// TwinCAT 3 PLC project JOGAN
// ProgramVersion: 3.1.4020.4
// libraries:
//   Tc2_Standard, * (Beckhoff Automation GmbH)
//   Tc2_System, * (Beckhoff Automation GmbH)
//   Tc3_Module, * (Beckhoff Automation GmbH)
// project tree:
//   DUTs/ T_CURRENT_TRANSACTION.TcDUT, T_JIG_SOCKET.TcDUT
//   GVLs/ FLAG_VAR.TcGVL, INDEXING_1_VAR.TcGVL, INDEXING_2_VAR.TcGVL, INPUT_G6_VAR.TcGVL, INPUT_VAR.TcGVL, LOADER_RS4_VAR.TcGVL, LOADER_VAR.TcGVL, POWER_CONTROL.TcGVL (not stored), SORTER_RS4_VAR.TcGVL, SORTER_VAR.TcGVL, TESTER_C8_VAR.TcGVL
//   / PlcTask.TcTTO
//   POUs/ EXECUTE_FUNCTION.TcPOU, INPUT_PROG.TcPOU, MAIN.TcPOU, STQWE.TcPOU (not stored)
//   POUs/FUKUDA/ FUKUDA_MOVE.TcPOU, FUKUDA_MOVE_1.TcPOU, LOAD_FUKUDA.TcPOU, LOAD_FUKUDA_1.TcPOU (not stored), RETURN_FUKUDA.TcPOU, RETURN_FUKUDA_1.TcPOU
//   POUs/LASER/ LASER_MOVE.TcPOU, LOAD_LASER.TcPOU, LOAD_NG.TcPOU, POU.TcPOU, RETURN_LASER.TcPOU, RETURN_NG.TcPOU
//   POUs/LOADER/ INDEXING.TcPOU, INDEX_1.TcPOU (not stored), INDEXING_2.TcPOU, STRAIGHTENING_PROG_1.TcPOU, STR.TcPOU
//   POUs/ROBOT/ INPUT_G6.TcPOU, INPUT_G61.TcPOU, LOADER_RS4.TcPOU, SORTER_RS4.TcPOU
// real-time tasks:
//   TASK PlcTask: cycle T#10ms, priority 20, ADS port 350
// I/O:
//   DEVICE Device 5 (EtherCAT), AmsNetId 172.18.128.227.6.1
//     Term 1 (EK1100) [EK1100 EtherCAT Coupler (2A E-Bus)]
//       Term 2 (EL1808) [EL1808 8Ch. Dig. Input 24V, 3ms]
//       Term 3 (EL1808) [EL1808 8Ch. Dig. Input 24V, 3ms]
//       Term 4 (EL1808) [EL1808 8Ch. Dig. Input 24V, 3ms]
//       Term 5 (EL1808) [EL1808 8Ch. Dig. Input 24V, 3ms]
//       Term 6 (EL2808) [EL2808 8Ch. Dig. Output 24V, 0.5A]
//       Term 7 (EL2808) [EL2808 8Ch. Dig. Output 24V, 0.5A]
//       Term 8 (EL2808) [EL2808 8Ch. Dig. Output 24V, 0.5A]
//       Term 9 (EL2808) [EL2808 8Ch. Dig. Output 24V, 0.5A]
//       Term 10 (EL2808) [EL2808 8Ch. Dig. Output 24V, 0.5A]
//       Term 11 (EL3058) [EL3058 8Ch. Ana. Input 4-20mA]
//       Term 12 (EL1904) [EL1904, 4 Ch. Safety Input 24V, TwinSAFE]
//         modules: Module 1 (FSOES)
//       Term 13 (EL1904) [EL1904, 4 Ch. Safety Input 24V, TwinSAFE]
//         modules: Module 1 (FSOES)
//       Term 14 (EL6731) [EL6731 PROFIBUS DP Master]
//       Term 15 (EK1110) [EK1110 EtherCAT extension]
//     Term 16 (EK1100) [EK1100 EtherCAT Coupler (2A E-Bus)]
//       Term 17 (EL1808) [EL1808 8Ch. Dig. Input 24V, 3ms]
//       Term 18 (EL1808) [EL1808 8Ch. Dig. Input 24V, 3ms]
//       Term 19 (EL1808) [EL1808 8Ch. Dig. Input 24V, 3ms]
//       Term 20 (EL1808) [EL1808 8Ch. Dig. Input 24V, 3ms]
//       Term 21 (EL1808) [EL1808 8Ch. Dig. Input 24V, 3ms]
//       Term 22 (EL1808) [EL1808 8K. Dig. Eingang 24V, 3ms]
//       Term 23 (EL2808) [EL2808 8Ch. Dig. Output 24V, 0.5A]
//       Term 24 (EL2808) [EL2808 8Ch. Dig. Output 24V, 0.5A]
//       Term 25 (EL2808) [EL2808 8Ch. Dig. Output 24V, 0.5A]
//       Term 26 (EL2808) [EL2808 8Ch. Dig. Output 24V, 0.5A]
//       Term 27 (EL2808) [EL2808 8Ch. Dig. Output 24V, 0.5A]
//       Term 28 (EL2808) [EL2808 8Ch. Dig. Output 24V, 0.5A]
//       Term 29 (EL2808) [EL2808 8Ch. Dig. Output 24V, 0.5A]
//       Term 30 (EL2808) [EL2808 8Ch. Dig. Output 24V, 0.5A]
//       Term 31 (EL6731) [EL6731 PROFIBUS DP Master]
//       Term 32 (EK1110) [EK1110 EtherCAT extension]
//     Box 33 (EP2809-0021)RS4-2 [EP2809-0021 16 Ch. Dig. Output 24V, 0,5A, M8]
//     Box 34 (EP1809-0021) [EP1809-0021 16 Ch. Dig. Input 24V, 3ms, M8]
//     Box 35 (EP2809-0021)RS4-1 [EP2809-0021 16 Ch. Dig. Output 24V, 0,5A, M8]
//     Box 36 (EP2809-0021)RS4-1 [EP1809-0021 16 Ch. Dig. Input 24V, 3ms, M8]
//     Box 37 (EP1809-0021) [EP1809-0021 16 Ch. Dig. Input 24V, 3ms, M8]
//     Box 38 (EP2809-0021) G6 [EP2809-0021 16 Ch. Dig. Output 24V, 0,5A, M8]
//     Box 39 (EPSON RC700 EtherCAT Slave)G6 [EPSON RC700 EtherCAT Slave]
//     Box 40 (EPSON RC700 EtherCAT Slave)RS4-1 [EPSON RC700 EtherCAT Slave]
//     Box 40 (EPSON RC700 EtherCAT Slave)C8 [EPSON RC700 EtherCAT Slave] (disabled)
//     Box 88 (EP2339-0021) [EP2339-0021 16 Ch. Dig. Input/Output 24V, 0,5A, M8] (disabled)
//     Box 42 (EPSON RC700 EtherCAT Slave)RS4-2 [EPSON RC700 EtherCAT Slave]
//   DEVICE Device 1 (EL6731), AmsNetId 172.18.128.227.2.1
//     Box 43 (LEC-GPR1) // Vendor: SMC Corporation Revision: V1.0
//     Box 44 (AX9000T) INDEXING 1 // Vendor: CKD Corporation Revision: Version 1.000
//      // Vendor: CKD Corporation Revision: Version 1.000
//   DEVICE Device 2 (EL6731), AmsNetId 172.18.128.227.3.1
//     Box 46 (LEC-GPR1) // Vendor: SMC Corporation Revision: V1.0
// variable links:
//   JOGAN/JOGAN Instance <-> Device 1 (EL6731)/
//     PlcTask Inputs/INDEXING_2_VAR.DataByteInput2 <-> Module 1 (8 Bytes Out,8 Bytes In)/Inputs/8 Bytes Out,8 Bytes In_0_0
//     PlcTask Outputs/INDEXING_2_VAR.DataByteOutput2 <-> Module 1 (8 Bytes Out,8 Bytes In)/Outputs/8 Bytes Out,8 Bytes In_1_0
//   JOGAN/JOGAN Instance <-> Device 1 (EL6731)/Box 43 (LEC-GPR1)
//     PlcTask Inputs/INPUT_VAR.DataWordInput1 <-> Module 1 (Input 16 words)/Inputs/Input 16 words_0_0
//     PlcTask Inputs/INPUT_VAR.DataWordInput2 <-> Module 2 (Input 16 words)/Inputs/Input 16 words_0_0
//     PlcTask Inputs/INPUT_VAR.DataWordInput3 <-> Module 3 (Input 16 words)/Inputs/Input 16 words_0_0
//     PlcTask Outputs/INPUT_VAR.DataWordOutput1 <-> Module 5 (Output 16 words)/Outputs/Output 16 words_1_0
//     PlcTask Outputs/INPUT_VAR.DataWordOutput2 <-> Module 6 (Output 16 words)/Outputs/Output 16 words_1_0
//     PlcTask Outputs/INPUT_VAR.DataWordOutput3 <-> Module 7 (Output 16 words)/Outputs/Output 16 words_1_0
//     PlcTask Outputs/INPUT_VAR.DataWordOutput4 <-> Module 8 (Output 9 words)/Outputs/Output 9 words_1_0
//   JOGAN/JOGAN Instance <-> Device 1 (EL6731)/Box 44 (AX9000T) INDEXING 1
//     PlcTask Inputs/INDEXING_1_VAR.DataByteInput <-> Module 2 (8 Bytes Out,8 Bytes In)/Inputs/8 Bytes Out,8 Bytes In_0_0
//     PlcTask Outputs/INDEXING_1_VAR.DataByteOutput <-> Module 2 (8 Bytes Out,8 Bytes In)/Outputs/8 Bytes Out,8 Bytes In_1_0
//   JOGAN/JOGAN Instance <-> Device 2 (EL6731)/Box 46 (LEC-GPR1)
//     PlcTask Inputs/SORTER_VAR.DataWordInput1 <-> Module 1 (Input 16 words)/Inputs/Input 16 words_0_0
//     PlcTask Inputs/SORTER_VAR.DataWordInput2 <-> Module 2 (Input 16 words)/Inputs/Input 16 words_0_0
//     PlcTask Inputs/SORTER_VAR.DataWordInput3 <-> Module 3 (Input 16 words)/Inputs/Input 16 words_0_0
//     PlcTask Inputs/SORTER_VAR.DataWordInput4 <-> Module 4 (Input 9 words)/Inputs/Input 9 words_0_0
//     PlcTask Outputs/SORTER_VAR.DataWordOutput1 <-> Module 5 (Output 16 words)/Outputs/Output 16 words_1_0
//     PlcTask Outputs/SORTER_VAR.DataWordOutput2 <-> Module 6 (Output 16 words)/Outputs/Output 16 words_1_0
//     PlcTask Outputs/SORTER_VAR.DataWordOutput3 <-> Module 7 (Output 16 words)/Outputs/Output 16 words_1_0
//     PlcTask Outputs/SORTER_VAR.DataWordOutput4 <-> Module 8 (Output 9 words)/Outputs/Output 9 words_1_0
//   JOGAN/JOGAN Instance <-> Device 5 (EtherCAT)/Box 33 (EP2809-0021)RS4-2
//     PlcTask Outputs/SORTER_RS4_VAR.O_SORTER_RS4_GRIPPER_CLOSE_{1..4} <-> Channel {1..7 step 2}/Output  (4 links)
//     PlcTask Outputs/SORTER_RS4_VAR.O_SORTER_RS4_GRIPPER_EXT_DOWN_{1..4} <-> Channel {9..15 step 2}/Output  (4 links)
//     PlcTask Outputs/SORTER_RS4_VAR.O_SORTER_RS4_GRIPPER_EXT_UP_{1..4} <-> Channel {10..16 step 2}/Output  (4 links)
//     PlcTask Outputs/SORTER_RS4_VAR.O_SORTER_RS4_GRIPPER_OPEN_{1..4} <-> Channel {2..8 step 2}/Output  (4 links)
//   JOGAN/JOGAN Instance <-> Device 5 (EtherCAT)/Box 35 (EP2809-0021)RS4-1
//     PlcTask Outputs/LOADER_RS4_VAR.O_LOADER_RS4_GRIPPER_CLOSE_{1..4} <-> Channel {1..7 step 2}/Output  (4 links)
//     PlcTask Outputs/LOADER_RS4_VAR.O_LOADER_RS4_GRIPPER_EXT_DOWN_{1..4} <-> Channel {9..15 step 2}/Output  (4 links)
//     PlcTask Outputs/LOADER_RS4_VAR.O_LOADER_RS4_GRIPPER_EXT_UP_{1..4} <-> Channel {10..16 step 2}/Output  (4 links)
//     PlcTask Outputs/LOADER_RS4_VAR.O_LOADER_RS4_GRIPPER_OPEN_{1..4} <-> Channel {2..8 step 2}/Output  (4 links)
//   JOGAN/JOGAN Instance <-> Device 5 (EtherCAT)/Box 38 (EP2809-0021) G6
//     PlcTask Outputs/INPUT_G6_VAR.O_G6_GRIPPER_CLOSE_{1..4} <-> Channel {1..7 step 2}/Output  (4 links)
//     PlcTask Outputs/INPUT_G6_VAR.O_G6_GRIPPER_EXT_DOWN_{1..4} <-> Channel {9..15 step 2}/Output  (4 links)
//     PlcTask Outputs/INPUT_G6_VAR.O_G6_GRIPPER_EXT_UP_{1..4} <-> Channel {10..16 step 2}/Output  (4 links)
//     PlcTask Outputs/INPUT_G6_VAR.O_G6_GRIPPER_OPEN_{1..4} <-> Channel {2..8 step 2}/Output  (4 links)
//   JOGAN/JOGAN Instance <-> Device 5 (EtherCAT)/Box 39 (EPSON RC700 EtherCAT Slave)G6
//     PlcTask Inputs/INPUT_G6_VAR.G6_INPUT <-> TxPDO/Input byte 0000
//     PlcTask Inputs/INPUT_G6_VAR.G6_INPUT_1 <-> TxPDO/Input byte 0001
//     PlcTask Inputs/INPUT_G6_VAR.G6_INPUT_2 <-> TxPDO/Input byte 0004
//     PlcTask Inputs/INPUT_G6_VAR.G6_INPUT_3 <-> TxPDO/Input byte 0005
//     PlcTask Outputs/INPUT_G6_VAR.G6_OUTPUT <-> RxPDO/Output byte 0000
//     PlcTask Outputs/INPUT_G6_VAR.G6_OUTPUT_1 <-> RxPDO/Output byte 0001
//     PlcTask Outputs/INPUT_G6_VAR.G6_OUTPUT_2 <-> RxPDO/Output byte 0002
//   JOGAN/JOGAN Instance <-> Device 5 (EtherCAT)/Box 40 (EPSON RC700 EtherCAT Slave)RS4-1
//     PlcTask Inputs/LOADER_RS4_VAR.LOADER_RS4_INPUT <-> TxPDO/Input byte 0000
//     PlcTask Inputs/LOADER_RS4_VAR.LOADER_RS4_INPUT_1 <-> TxPDO/Input byte 0001
//     PlcTask Inputs/LOADER_RS4_VAR.LOADER_RS4_INPUT_2 <-> TxPDO/Input byte 0004
//     PlcTask Inputs/LOADER_RS4_VAR.LOADER_RS4_INPUT_3 <-> TxPDO/Input byte 0005
//     PlcTask Outputs/LOADER_RS4_VAR.CARRIER_INDEX <-> RxPDO/Output byte 0006
//     PlcTask Outputs/LOADER_RS4_VAR.LOADER_RS4_OUTPUT <-> RxPDO/Output byte 0000
//     PlcTask Outputs/LOADER_RS4_VAR.LOADER_RS4_OUTPUT_1 <-> RxPDO/Output byte 0001
//     PlcTask Outputs/LOADER_RS4_VAR.LOADER_RS4_OUTPUT_2 <-> RxPDO/Output byte 0002
//     PlcTask Outputs/LOADER_RS4_VAR.LOADER_RS4_OUTPUT_3 <-> RxPDO/Output byte 0003
//     PlcTask Outputs/LOADER_RS4_VAR.LOADER_RS4_OUTPUT_4 <-> RxPDO/Output byte 0004
//     PlcTask Outputs/LOADER_RS4_VAR.LOADER_RS4_OUTPUT_5 <-> RxPDO/Output byte 0005
//   JOGAN/JOGAN Instance <-> Device 5 (EtherCAT)/Box 42 (EPSON RC700 EtherCAT Slave)RS4-2
//     PlcTask Inputs/SORTER_RS4_VAR.SORTER_RS4_INPUT <-> TxPDO/Input byte 0000
//     PlcTask Inputs/SORTER_RS4_VAR.SORTER_RS4_INPUT_1 <-> TxPDO/Input byte 0001
//     PlcTask Inputs/SORTER_RS4_VAR.SORTER_RS4_INPUT_2 <-> TxPDO/Input byte 0004
//     PlcTask Inputs/SORTER_RS4_VAR.SORTER_RS4_INPUT_3 <-> TxPDO/<empty>
//     PlcTask Outputs/SORTER_RS4_VAR.SORTER_RS4_OUTPUT <-> RxPDO/Output byte 0000
//     PlcTask Outputs/SORTER_RS4_VAR.SORTER_RS4_OUTPUT_1 <-> RxPDO/Output byte 0001
//     PlcTask Outputs/SORTER_RS4_VAR.SORTER_RS4_POS_PLACING_1 <-> RxPDO/Output byte 0006
//     PlcTask Outputs/SORTER_RS4_VAR.SORTER_RS4_POS_PLACING_2 <-> RxPDO/Output byte 0007
//     PlcTask Outputs/SORTER_RS4_VAR.SORTER_RS4_POS_PLACING_3 <-> RxPDO/Output byte 0008
//     PlcTask Outputs/SORTER_RS4_VAR.SORTER_RS4_POS_PLACING_4 <-> RxPDO/Output byte 0009
//     PlcTask Outputs/SORTER_RS4_VAR.SORTER_RS4_POS_TAKEUP_1 <-> RxPDO/Output byte 0002
//     PlcTask Outputs/SORTER_RS4_VAR.SORTER_RS4_POS_TAKEUP_2 <-> RxPDO/Output byte 0003
//     PlcTask Outputs/SORTER_RS4_VAR.SORTER_RS4_POS_TAKEUP_3 <-> RxPDO/Output byte 0004
//     PlcTask Outputs/SORTER_RS4_VAR.SORTER_RS4_POS_TAKEUP_4 <-> RxPDO/Output byte 0005
//   JOGAN/JOGAN Instance <-> Device 5 (EtherCAT)/Term 1 (EK1100)/Term 10 (EL2808)
//     PlcTask Outputs/INPUT_VAR.O_RESET_CARTESSIAN <-> Channel 3/Output
//     PlcTask Outputs/INPUT_VAR.O_STOPPER_TRANSFER_A <-> Channel 1/Output
//     PlcTask Outputs/INPUT_VAR.O_STOPPER_TRANSFER_B <-> Channel 2/Output
//   JOGAN/JOGAN Instance <-> Device 5 (EtherCAT)/Term 1 (EK1100)/Term 2 (EL1808)
//     PlcTask Inputs/INPUT_VAR.I_FUKUDA_TRANSFER_AT_BACK_A <-> Channel 3/Input
//     PlcTask Inputs/INPUT_VAR.I_FUKUDA_TRANSFER_AT_BACK_B <-> Channel 1/Input
//     PlcTask Inputs/INPUT_VAR.I_FUKUDA_TRANSFER_AT_FRONT_A <-> Channel 4/Input
//     PlcTask Inputs/INPUT_VAR.I_FUKUDA_TRANSFER_AT_FRONT_B <-> Channel 2/Input
//     PlcTask Inputs/INPUT_VAR.I_LOTBOX_DETECT_{1..4} <-> Channel {5..8}/Input  (4 links)
//   JOGAN/JOGAN Instance <-> Device 5 (EtherCAT)/Term 1 (EK1100)/Term 3 (EL1808)
//     PlcTask Inputs/INDEXING_1_VAR.I_INDEXING_1_GRIPPER_CLOSE_{1..4} <-> Channel {1..7 step 2}/Input  (4 links)
//     PlcTask Inputs/INDEXING_1_VAR.I_INDEXING_1_GRIPPER_OPEN_{1..4} <-> Channel {2..8 step 2}/Input  (4 links)
//   JOGAN/JOGAN Instance <-> Device 5 (EtherCAT)/Term 1 (EK1100)/Term 4 (EL1808)
//     PlcTask Inputs/INDEXING_1_VAR.I_INDEXING_1_GRIPPER_EXT_DOWN <-> Channel 2/Input
//     PlcTask Inputs/INDEXING_1_VAR.I_INDEXING_1_GRIPPER_EXT_UP <-> Channel 1/Input
//     PlcTask Inputs/INPUT_VAR.I_LOTBOX_CLAMP_OFF_1 <-> Channel 6/Input
//     PlcTask Inputs/INPUT_VAR.I_LOTBOX_CLAMP_OFF_2 <-> Channel 8/Input
//     PlcTask Inputs/INPUT_VAR.I_LOTBOX_CLAMP_ON_1 <-> Channel 5/Input
//     PlcTask Inputs/INPUT_VAR.I_LOTBOX_CLAMP_ON_2 <-> Channel 7/Input
//   JOGAN/JOGAN Instance <-> Device 5 (EtherCAT)/Term 1 (EK1100)/Term 5 (EL1808)
//     PlcTask Inputs/INDEXING_1_VAR.I_PRESS_STOPPER_DOWN <-> Channel 7/Input
//     PlcTask Inputs/INDEXING_1_VAR.I_PRESS_STOPPER_UP <-> Channel 8/Input
//     PlcTask Inputs/INPUT_VAR.I_LOTBOX_CLAMP_OFF_3 <-> Channel 2/Input
//     PlcTask Inputs/INPUT_VAR.I_LOTBOX_CLAMP_OFF_4 <-> Channel 4/Input
//     PlcTask Inputs/INPUT_VAR.I_LOTBOX_CLAMP_ON_3 <-> Channel 1/Input
//     PlcTask Inputs/INPUT_VAR.I_LOTBOX_CLAMP_ON_4 <-> Channel 3/Input
//     PlcTask Inputs/INPUT_VAR.I_VACUUM_OFF <-> Channel 6/Input
//     PlcTask Inputs/INPUT_VAR.I_VACUUM_ON <-> Channel 5/Input
//   JOGAN/JOGAN Instance <-> Device 5 (EtherCAT)/Term 1 (EK1100)/Term 6 (EL2808)
//     PlcTask Outputs/INPUT_VAR.O_VACUUM_OFF <-> Channel 2/Output
//     PlcTask Outputs/INPUT_VAR.O_VACUUM_ON <-> Channel 1/Output
//   JOGAN/JOGAN Instance <-> Device 5 (EtherCAT)/Term 1 (EK1100)/Term 7 (EL2808)
//     PlcTask Outputs/INDEXING_1_VAR.O_INDEXING_1_GRIPPER_CLOSE_{1..4} <-> Channel {1..7 step 2}/Output  (4 links)
//     PlcTask Outputs/INDEXING_1_VAR.O_INDEXING_1_GRIPPER_OPEN_{1..4} <-> Channel {2..8 step 2}/Output  (4 links)
//   JOGAN/JOGAN Instance <-> Device 5 (EtherCAT)/Term 1 (EK1100)/Term 8 (EL2808)
//     PlcTask Outputs/INDEXING_1_VAR.O_INDEXING_1_GRIPPER_EXT_DOWN <-> Channel 2/Output
//     PlcTask Outputs/INDEXING_1_VAR.O_INDEXING_1_GRIPPER_EXT_UP <-> Channel 1/Output
//     PlcTask Outputs/INDEXING_1_VAR.O_PRESS_STOPPER_DOWN <-> Channel 7/Output
//     PlcTask Outputs/INDEXING_1_VAR.O_PRESS_STOPPER_UP <-> Channel 8/Output
//   JOGAN/JOGAN Instance <-> Device 5 (EtherCAT)/Term 1 (EK1100)/Term 9 (EL2808)
//     PlcTask Outputs/INPUT_VAR.O_LOTBOX_CLAMP_OFF_{1..4} <-> Channel {7..1 step -2}/Output  (4 links)
//     PlcTask Outputs/INPUT_VAR.O_LOTBOX_CLAMP_ON_{1..4} <-> Channel {8..2 step -2}/Output  (4 links)
//   JOGAN/JOGAN Instance <-> Device 5 (EtherCAT)/Term 16 (EK1100)/Term 19 (EL1808)
//     PlcTask Inputs/SORTER_VAR.I_LASER_TRANSFER_AT_BACK_A <-> Channel 7/Input
//     PlcTask Inputs/SORTER_VAR.I_LASER_TRANSFER_AT_FRONT_A <-> Channel 6/Input
//     PlcTask Inputs/SORTER_VAR.I_LASER_TRANSFER_AT_FRONT_B <-> Channel 8/Input
//   JOGAN/JOGAN Instance <-> Device 5 (EtherCAT)/Term 16 (EK1100)/Term 20 (EL1808)
//     PlcTask Inputs/SORTER_VAR.I_LASER_TRANSFER_AT_BACK_B <-> Channel 1/Input
//     PlcTask Inputs/SORTER_VAR.I_NG_TRANSFER_AT_BACK <-> Channel 2/Input
//     PlcTask Inputs/SORTER_VAR.I_NG_TRANSFER_AT_FRONT <-> Channel 3/Input
//   JOGAN/JOGAN Instance <-> Device 5 (EtherCAT)/Term 16 (EK1100)/Term 23 (EL2808)
//     PlcTask Outputs/SORTER_VAR.O_LOTBOX_CLAMP_OFF_{1..4} <-> Channel {1..7 step 2}/Output  (4 links)
//     PlcTask Outputs/SORTER_VAR.O_LOTBOX_CLAMP_ON_{1..4} <-> Channel {2..8 step 2}/Output  (4 links)
//   JOGAN/JOGAN Instance <-> Device 5 (EtherCAT)/Term 16 (EK1100)/Term 24 (EL2808)
//     PlcTask Outputs/SORTER_VAR.O_VACUUM_OFF <-> Channel 4/Output
//     PlcTask Outputs/SORTER_VAR.O_VACUUM_ON <-> Channel 3/Output
//   JOGAN/JOGAN Instance <-> Device 5 (EtherCAT)/Term 16 (EK1100)/Term 26 (EL2808)
//     PlcTask Outputs/SORTER_VAR.O_NG_DATA_OUTPUT{1..4} <-> Channel {5..8}/Output  (4 links)
//   JOGAN/JOGAN Instance <-> Device 5 (EtherCAT)/Term 16 (EK1100)/Term 30 (EL2808)
//     PlcTask Outputs/INDEXING_2_VAR.O_INDEXING_2_POWER_OFF <-> Channel 8/Output

CONFIGURATION JOGAN
    RESOURCE PLC ON TwinCAT3
        TASK PlcTask(INTERVAL := T#10ms, PRIORITY := 20);
        PROGRAM MAIN WITH PlcTask : MAIN;
    END_RESOURCE
END_CONFIGURATION

// ---- DUTs/T_CURRENT_TRANSACTION.TcDUT
TYPE T_CURRENT_TRANSACTION :
STRUCT
	STATION_NUMBER_LOAD : BYTE :=4;
	STATION_NUMBER_RETURN : BYTE :=4;
	QUANTITY_MAX : BYTE :=0;
	QUANTITY_LOTEND :BYTE :=0;
	JIG_INDEX_LOAD : BYTE :=1;
	JIG_INDEX_RETURN : BYTE :=1;
	TRANSPORT_INDEX : BYTE :=1;
	PO_NUMBER : STRING[255] := '';
END_STRUCT
END_TYPE

// ---- DUTs/T_JIG_SOCKET.TcDUT
TYPE T_JIG_SOCKET :
STRUCT
	AVAILABLE_SOCKET : ARRAY[0..4] OF DINT;
	LASER_DESTINATION: ARRAY[0..4] OF DINT;
END_STRUCT
END_TYPE

// ---- GVLs/FLAG_VAR.TcGVL
{attribute 'qualified_only'}
VAR_GLOBAL
	ALLOW_EXECUTE_LOAD_FUKUDA : BOOL:=FALSE;
	ALLOW_EXECUTE_RETURN_FUKUDA:BOOL:=FALSE;

	ALLOW_EXECUTE_LOAD_LASER : BOOL:=FALSE;
	ALLOW_EXECUTE_RETURN_LASER:BOOL:=FALSE;
	
	ALLOW_EXECUTE_LOAD_NG : BOOL:=FALSE;
	ALLOW_EXECUTE_RETURN_NG:BOOL:=FALSE;
END_VAR

// ---- GVLs/INDEXING_1_VAR.TcGVL
{attribute 'qualified_CLOSEly'}
VAR_GLOBAL
	
I_INDEXING_1_GRIPPER_CLOSE_1 AT %I* : BOOL;
I_INDEXING_1_GRIPPER_CLOSE_2 AT %I* : BOOL;
I_INDEXING_1_GRIPPER_CLOSE_3 AT %I* : BOOL;
I_INDEXING_1_GRIPPER_CLOSE_4 AT %I* : BOOL;
I_INDEXING_1_GRIPPER_OPEN_1 AT %I* : BOOL;
I_INDEXING_1_GRIPPER_OPEN_2 AT %I* : BOOL;
I_INDEXING_1_GRIPPER_OPEN_3 AT %I* : BOOL;
I_INDEXING_1_GRIPPER_OPEN_4 AT %I* : BOOL;
I_INDEXING_1_GRIPPER_EXT_UP AT %I* : BOOL;
I_INDEXING_1_GRIPPER_EXT_DOWN AT %I* : BOOL;

O_INDEXING_1_GRIPPER_EXT_UP AT %Q* : BOOL;
O_INDEXING_1_GRIPPER_EXT_DOWN AT %Q* : BOOL;
O_INDEXING_1_GRIPPER_CLOSE_1 AT %Q* : BOOL;
O_INDEXING_1_GRIPPER_CLOSE_2 AT %Q* : BOOL;
O_INDEXING_1_GRIPPER_CLOSE_3 AT %Q* : BOOL;
O_INDEXING_1_GRIPPER_CLOSE_4 AT %Q* : BOOL;
O_INDEXING_1_GRIPPER_OPEN_1 AT %Q* : BOOL;
O_INDEXING_1_GRIPPER_OPEN_2 AT %Q* : BOOL;
O_INDEXING_1_GRIPPER_OPEN_3 AT %Q* : BOOL;
O_INDEXING_1_GRIPPER_OPEN_4 AT %Q* : BOOL;

I_PRESS_STOPPER_DOWN AT %I* : BOOL;
I_PRESS_STOPPER_UP AT %I* : BOOL;

O_PRESS_STOPPER_DOWN AT %Q* : BOOL;
O_PRESS_STOPPER_UP AT %Q* : BOOL;

O_INDEXING_1_HOME   : BOOL;
O_ROTATION_START : BOOL;
O_ROTATION_STOP : BOOL;

I_INDEXING_1_READY_FOR_STRAIGHTEN: BOOL;
I_INDEXING_1_HOME AT %I* : BOOL;
O_INDEXING_1_POWER_OFF AT %Q* : BOOL;

I_INDEXING_1_ROTATION_START: BOOL;
I_INDEXING_1_ROTATION_PROCESS: BOOL;
I_INDEXING_1_ROTATION_DONE: BOOL ;

I_ALL_GRIPPER_OPEN: BOOL;
NUMBER_OF_STRAIGHTEN: INT :=0;
INDEXING_1_CASE: INT ;
TOTALNUMBER_OF_STRAIGHTEN :INT :=1;
STRAIGHTEN_FINISH:BOOL;
READY_STRAIGTHEN: BOOL;

DataByteOutput AT%Q* : ARRAY[0..7] OF BYTE;
DataByteInput AT%I* : ARRAY[0..7] OF BYTE;
END_VAR

// ---- GVLs/INDEXING_2_VAR.TcGVL
{attribute 'qualified_CLOSEly'}
VAR_GLOBAL
	
I_INDEXING_22_GRIPPER_CLOSE_1 AT %I* : BOOL;
I_INDEXING_2_GRIPPER_CLOSE_2 AT %I* : BOOL;
I_INDEXING_2_GRIPPER_CLOSE_3 AT %I* : BOOL;
I_INDEXING_2_GRIPPER_CLOSE_4 AT %I* : BOOL;
I_INDEXING_2_GRIPPER_OPEN_1 AT %I* : BOOL;
I_INDEXING_2_GRIPPER_OPEN_2 AT %I* : BOOL;
I_INDEXING_2_GRIPPER_OPEN_3 AT %I* : BOOL;
I_INDEXING_2_GRIPPER_OPEN_4 AT %I* : BOOL;
I_INDEXING_2_GRIPPER_EXT_UP AT %I* : BOOL;
I_INDEXING_2_GRIPPER_EXT_DOWN AT %I* : BOOL;

O_INDEXING_2_GRIPPER_EXT_UP AT %Q* : BOOL;
O_INDEXING_2_GRIPPER_EXT_DOWN AT %Q* : BOOL;
O_INDEXING_2_GRIPPER_CLOSE_1 AT %Q* : BOOL;
O_INDEXING_2_GRIPPER_CLOSE_2 AT %Q* : BOOL;
O_INDEXING_2_GRIPPER_CLOSE_3 AT %Q* : BOOL;
O_INDEXING_2_GRIPPER_CLOSE_4 AT %Q* : BOOL;
O_INDEXING_2_GRIPPER_OPEN_1 AT %Q* : BOOL;
O_INDEXING_2_GRIPPER_OPEN_2 AT %Q* : BOOL;
O_INDEXING_2_GRIPPER_OPEN_3 AT %Q* : BOOL;
O_INDEXING_2_GRIPPER_OPEN_4 AT %Q* : BOOL;

I_PRESS_STOPPER_DOWN AT %I* : BOOL;
I_PRESS_STOPPER_UP AT %I* : BOOL;

O_PRESS_STOPPER_DOWN AT %Q* : BOOL;
O_PRESS_STOPPER_UP AT %Q* : BOOL;

O_INDEXING_HOME   : BOOL;
O_ROTATION_DONE : BOOL;
O_ROTATION_START : BOOL;
O_ROTATION_STOP : BOOL;

I_INDEXING_2_READY_FOR_STRAIGHTEN: BOOL;
I_INDEXING_2_HOME AT %Q* : BOOL;
O_INDEXING_2_POWER_OFF AT %Q* : BOOL;

I_INDEXING_2_ROTATION_DONE: BOOL :=TRUE;
I_ALL_GRIPPER_OPEN: BOOL;
NUMBER_OF_STRAIGHTEN: INT :=0;
INDEXING_2_CASE: INT ;
TOTALNUMBER_OF_STRAIGHTEN :INT :=1;
CARRIER_INDEX: BYTE;

DataByteOutput2 AT%Q* : ARRAY[0..7] OF BYTE;
DataByteInput2 AT%I* : ARRAY[0..7] OF BYTE;
END_VAR

// ---- GVLs/INPUT_G6_VAR.TcGVL
{attribute 'qualified_only'}
VAR_GLOBAL
G6_INPUT AT %IB00 :  	BYTE;
G6_INPUT_1 AT %IB01 : 	BYTE;
G6_INPUT_2 AT %IB02 : 	BYTE;
G6_INPUT_3 AT %IB03 :	BYTE;
G6_OUTPUT AT %QB00 : 	BYTE;
G6_OUTPUT_1 AT %QB01 : BYTE;
G6_OUTPUT_2 AT %QB02 : BYTE;

I_G6_READY  AT %IX0.0 :BOOL;
I_G6_RUNNING  AT %IX0.1 :BOOL;
I_G6_PAUSED  AT %IX0.2 :BOOL;
I_G6_ERROR  AT %IX0.3 :BOOL;
I_G6_ESTOPON  AT %IX0.4 :BOOL;
I_G6_SAFEGUARDON  AT %IX0.5 :BOOL;
I_G6_SERROR  AT %IX0.6 :BOOL;
I_G6_WARNING  AT %IX0.7 :BOOL;

I_G6_MOTORON  AT %IX1.0 :BOOL;
I_G6_ATHOME  AT %IX1.1 :BOOL;
I_G6_AUTOMODE  AT %IX1.5 :BOOL;
	
I_G6_END_CYCLE  AT %IX3.0 :BOOL;
I_G6_END_FUKUDA  AT %IX3.1 :BOOL;
I_G6_READY_TAKEUP  AT %IX3.2 :BOOL;//CYCLE RUNNING INDICATOR
I_G6_START_TAKEUP  AT %IX3.3 :BOOL;
I_G6_READY_PLACING  AT %IX3.4 :BOOL;
I_G6_START_PLACING  AT %IX3.5 :BOOL;
	
	O_G6_START AT %QX00.0  : BOOL;	
	O_G6_SELECT_FUKUDA_A AT %QX00.1  : BOOL;
	O_G6_SELECT_FUKUDA_B AT %QX00.2  : BOOL;
	O_G6_STOP AT %QX00.4  : BOOL;
	O_G6_PAUSE AT %QX00.5  : BOOL;
	O_G6_CONTINUE AT %QX00.6  : BOOL;
	O_G6_RESET AT %QX00.7  : BOOL;	
	
	O_G6_SETMOTORON AT %QX01.0  : BOOL;
	O_G6_SETMOTOROFF AT %QX01.1  : BOOL;
	O_G6_HOME AT %QX01.2  : BOOL;
		
I_G6_GRIPPER_CLOSE_1 AT %I* : BOOL;
I_G6_GRIPPER_CLOSE_2 AT %I* : BOOL;
I_G6_GRIPPER_CLOSE_3 AT %I* : BOOL;
I_G6_GRIPPER_CLOSE_4 AT %I* : BOOL;
I_G6_GRIPPER_OPEN_1 AT %I* : BOOL;
I_G6_GRIPPER_OPEN_2 AT %I* : BOOL;
I_G6_GRIPPER_OPEN_3 AT %I* : BOOL;
I_G6_GRIPPER_OPEN_4 AT %I* : BOOL;
I_G6_GRIPPER_EXT_DOWN_1 AT %I* : BOOL;
I_G6_GRIPPER_EXT_DOWN_2 AT %I* : BOOL;
I_G6_GRIPPER_EXT_DOWN_3 AT %I* : BOOL;
I_G6_GRIPPER_EXT_DOWN_4 AT %I* : BOOL;
I_G6_GRIPPER_EXT_UP_1 AT %I* : BOOL;
I_G6_GRIPPER_EXT_UP_2 AT %I* : BOOL;
I_G6_GRIPPER_EXT_UP_3 AT %I* : BOOL;
I_G6_GRIPPER_EXT_UP_4 AT %I* : BOOL;

	O_G6_GRIPPER_CLOSE_1 AT %Q* : BOOL;
	O_G6_GRIPPER_CLOSE_2 AT %Q* : BOOL;
	O_G6_GRIPPER_CLOSE_3 AT %Q* : BOOL;
	O_G6_GRIPPER_CLOSE_4 AT %Q* : BOOL;
	O_G6_GRIPPER_OPEN_1 AT %Q* : BOOL;
	O_G6_GRIPPER_OPEN_2 AT %Q* : BOOL;
	O_G6_GRIPPER_OPEN_3 AT %Q* : BOOL;
	O_G6_GRIPPER_OPEN_4 AT %Q* : BOOL;
	O_G6_GRIPPER_EXT_DOWN_1 AT %Q* : BOOL;
	O_G6_GRIPPER_EXT_DOWN_2 AT %Q* : BOOL;
	O_G6_GRIPPER_EXT_DOWN_3 AT %Q* : BOOL;
	O_G6_GRIPPER_EXT_DOWN_4 AT %Q* : BOOL;
	O_G6_GRIPPER_EXT_UP_1 AT %Q* : BOOL;
	O_G6_GRIPPER_EXT_UP_2 AT %Q* : BOOL;
	O_G6_GRIPPER_EXT_UP_3 AT %Q* : BOOL;
	O_G6_GRIPPER_EXT_UP_4 AT %Q* : BOOL;

IX_G6_GRIPPER_1 AT %IX2.0 : BOOL;
IX_G6_GRIPPER_2 AT %IX2.1 : BOOL;
IX_G6_GRIPPER_3 AT %IX2.2 : BOOL;
IX_G6_GRIPPER_4 AT %IX2.3 : BOOL;

IX_G6_GRIPPER_EXT_1 AT %IX2.4 : BOOL;
IX_G6_GRIPPER_EXT_2 AT %IX2.5 : BOOL;
IX_G6_GRIPPER_EXT_3 AT %IX2.6 : BOOL;
IX_G6_GRIPPER_EXT_4 AT %IX2.7 : BOOL;

	OX_G6_GRIPPER_1 AT %QX02.0 : BOOL;
	OX_G6_GRIPPER_2 AT %QX02.1 : BOOL;
	OX_G6_GRIPPER_3 AT %QX02.2 : BOOL;
	OX_G6_GRIPPER_4 AT %QX02.3 : BOOL;

	OX_G6_GRIPPER_EXT_1 AT %QX02.4 : BOOL;
	OX_G6_GRIPPER_EXT_2 AT %QX02.5 : BOOL;
	OX_G6_GRIPPER_EXT_3 AT %QX02.6 : BOOL;
	OX_G6_GRIPPER_EXT_4 AT %QX02.7 : BOOL;

IX_G6_FINISH AT %I* : BOOL;
I_G6_HANG : BOOL;
I_G6_ENABLE :BOOL;
I_G6_DISABLE :BOOL;
GO_ROBOT :BOOL;
	
		
END_VAR

// ---- GVLs/INPUT_VAR.TcGVL
{attribute 'qualified_only'}
VAR_GLOBAL
I_LOTBOX_CLAMP_ON_1 AT %I* : BOOL;
I_LOTBOX_CLAMP_ON_2 AT %I* : BOOL;
I_LOTBOX_CLAMP_ON_3 AT %I* : BOOL;
I_LOTBOX_CLAMP_ON_4 AT %I* : BOOL;
I_LOTBOX_CLAMP_OFF_1 AT %I* : BOOL;
I_LOTBOX_CLAMP_OFF_2 AT %I* : BOOL;
I_LOTBOX_CLAMP_OFF_3 AT %I* : BOOL;
I_LOTBOX_CLAMP_OFF_4 AT %I* : BOOL;
	
I_LOTBOX_DETECT_1 AT %I* : BOOL;//LOTBOX_FUKUDA1_DETECT
I_LOTBOX_DETECT_2 AT %I* : BOOL;//LOTBOX_FUKUDA2_DETECT
I_LOTBOX_DETECT_3 AT %I* : BOOL;//LOTBOX_FUKUDA3_DETECT
I_LOTBOX_DETECT_4 AT %I* : BOOL;//LOTBOX_FUKUDA4_DETECT

I_VACUUM_ON AT %I* : BOOL;
I_VACUUM_OFF AT %I* : BOOL;

I_FUKUDA_TRANSFER_AT_FRONT_A AT %I* : BOOL;
I_FUKUDA_TRANSFER_AT_BACK_A AT %I* : BOOL;
I_FUKUDA_TRANSFER_AT_FRONT_B AT %I* : BOOL;
I_FUKUDA_TRANSFER_AT_BACK_B AT %I* : BOOL;
I_FUKUDA_TRANSFER_A_PICK_DONE : BOOL;
I_FUKUDA_TRANSFER_B_PICK_DONE : BOOL;
I_FUKUDA_TRANSFER_AT_A : BOOL;
I_FUKUDA_TRANSFER_AT_B : BOOL;

I_RETURN_DONE_A: BOOL;
I_RETURN_DONE_B: BOOL;
I_LOADING_DONE_A: BOOL;
I_LOADING_DONE_B: BOOL;
I_CURRENT_TRANSACTION : T_CURRENT_TRANSACTION ;
I_FUKUDA_ONDUTY_A:BOOL;
I_FUKUDA_ONDUTY_B:BOOL;
JIG_FUKUDA_PRESENCE: BOOL :=TRUE;

I_LOTEND :BOOL :=TRUE;
I_FUNC_CALLED:BOOL:=TRUE;
I_LOADING_DONE : BOOL;
I_LOADING_FAILED: BOOL;
I_LOADING_ALARM: INT;
I_LOADING_SOCKET : T_JIG_SOCKET;
I_LASER_SOCKET : T_JIG_SOCKET; 
I_CARTESSIAN_GRIPPER_ON AT %I* : BOOL;
I_CARTESSIAN_GRIPPER_OFF AT %I* : BOOL;
I_FUNCTION_NAME :STRING [255];
I_CASE : INT:=0;
I_FUKUDA_RUNNING:BOOL :=FALSE;

O_LOTBOX_CLAMP_ON_1 AT %Q* : BOOL;
O_LOTBOX_CLAMP_ON_2 AT %Q* : BOOL;
O_LOTBOX_CLAMP_ON_3 AT %Q* : BOOL;
O_LOTBOX_CLAMP_ON_4 AT %Q* : BOOL;
O_LOTBOX_CLAMP_OFF_1 AT %Q* : BOOL;
O_LOTBOX_CLAMP_OFF_2 AT %Q* : BOOL;
O_LOTBOX_CLAMP_OFF_3 AT %Q* : BOOL;
O_LOTBOX_CLAMP_OFF_4 AT %Q* : BOOL;

O_VACUUM_ON AT %Q* : BOOL;
O_VACUUM_OFF AT %Q* : BOOL;
O_CARTESSIAN_GRIPPER_ON AT %Q* : BOOL;
O_CARTESSIAN_GRIPPER_OFF AT %Q* : BOOL;
O_TOWER_LAMP_RED AT %Q* : BOOL;
O_TOWER_LAMP_YELLOW AT %Q* : BOOL;
O_TOWER_LAMP_GREEN AT %Q* : BOOL;
O_TOWER_LAMP_BUZZER AT %Q* : BOOL;
O_WARNING_LIGHT AT %Q* : BOOL;
O_LOT_BOX_INDICATOR_1  AT %Q* : BOOL;
O_LOT_BOX_INDICATOR_2 AT %Q* : BOOL;
O_LOT_BOX_INDICATOR_3 AT %Q* : BOOL;
O_LOT_BOX_INDICATOR_4 AT %Q* : BOOL;

AXIS_COMPLETE: BOOL;
LOTBOX_READY_1: BOOL;

DataWordInput1 AT %IB100 : ARRAY [0..15] OF WORD; 
DataWordInput2 AT %IB132 : ARRAY [16..31] OF WORD; 
DataWordInput3 AT %IB164 : ARRAY [32..47] OF WORD; 
DataWordInput4 AT %IB196 : ARRAY [48..56] OF WORD; 
DataWordOutput1 AT %QB100 : ARRAY [0..15] OF WORD; 
DataWordOutput2 AT %QB132 : ARRAY [16..31] OF WORD; 
DataWordOutput3 AT %QB164 : ARRAY [32..47] OF WORD; 
DataWordOutput4 AT %QB196 : ARRAY [48..56] OF WORD; 

I_RETURN_ALARM: INT;
I_RETURN_FAILED: BOOL;
ACTIVE_ID: INT :=1;	
ACTIVE_PROGRAM: INT ;
ACTIVE_PROGRAM_CHANGE:BOOL;
	
I_FUKUDA_HOME : BOOL;
O_FUKUDA_HOME : BOOL; 
STRAIGHTEN_START: BOOL;
STRAIGHTEN_PROCESS: BOOL;
STRAIGHTEN_DONE: BOOL;

FUKUDA_HOME: BOOL;

O_STOPPER_TRANSFER_A AT %Q* : BOOL;
O_STOPPER_TRANSFER_B AT %Q* : BOOL;
I_STOPPER_TRANSFER_ON_A AT %Q* : BOOL;
I_STOPPER_TRANSFER_OFF_A AT %Q* : BOOL;
I_STOPPER_TRANSFER_ON_B AT %Q* : BOOL;
I_STOPPER_TRANSFER_OFF_B AT %Q* : BOOL;
O_RESET_CARTESSIAN AT %Q* : BOOL;

END_VAR

// ---- GVLs/LOADER_RS4_VAR.TcGVL
{attribute 'qualified_only'}
VAR_GLOBAL

LOADER_RS4_INPUT AT %IB32 : ARRAY [0..15] OF WORD; 
LOADER_RS4_INPUT_1 AT %IB33 : ARRAY [0..15] OF WORD;
LOADER_RS4_INPUT_2 AT %IB36 : ARRAY [0..15] OF WORD;
LOADER_RS4_INPUT_3 AT %IB37 : ARRAY [0..15] OF WORD;
LOADER_RS4_OUTPUT AT %QB32 : ARRAY [0..15] OF WORD;
LOADER_RS4_OUTPUT_1 AT %QB33 : ARRAY [0..15] OF WORD;
LOADER_RS4_OUTPUT_2 AT %QB34 : BYTE :=1;
LOADER_RS4_OUTPUT_3 AT %QB35 : BYTE :=2;
LOADER_RS4_OUTPUT_4 AT %QB36 : BYTE :=3;
LOADER_RS4_OUTPUT_5 AT %QB37 : BYTE :=4;
CARRIER_INDEX AT %QB38 : BYTE ;

I_LOADER_RS4_READY  AT %IX32.0 :BOOL;
I_LOADER_RS4_RUNNING  AT %IX32.1 :BOOL;
I_LOADER_RS4_PAUSED  AT %IX32.2 :BOOL;
I_LOADER_RS4_ERROR  AT %IX32.3 :BOOL;
I_LOADER_RS4_ESTOPON  AT %IX32.4 :BOOL;
I_LOADER_RS46_SAFEGUARDON  AT %IX32.5 :BOOL;
I_LOADER_RS4_SERROR  AT %IX32.6 :BOOL;
I_LOADER_RS4_WARNING  AT %IX32.7 :BOOL;

I_LOADER_RS4_MOTORON  AT %IX33.0 :BOOL;
I_LOADER_RS4_ATHOME  AT %IX33.1 :BOOL;
I_LOADER_RS4_AUTOMODE  AT %IX33.5 :BOOL;
	
I_LOADER_RS4_END_CYCLE  AT %IX37.0 :BOOL;
I_LOADER_RS4_END_FUKUDA  AT %IX37.1 :BOOL;
I_LOADER_RS4_READY_TAKEUP  AT %IX37.2 :BOOL;//CYCLE RUNNING INDICATOR
I_LOADER_RS4_START_TAKEUP  AT %IX37.3 :BOOL;
I_LOADER_RS4_READY_PLACING  AT %IX37.4 :BOOL;
I_LOADER_RS4_START_PLACING  AT %IX37.5 :BOOL;
	
	O_LOADER_RS4_START AT %QX32.0  : BOOL;	
	O_LOADER_RS4_SELECT_FUKUDA_A AT %QX32.1  : BOOL;
	O_LOADER_RS4_SELECT_FUKUDA_B AT %QX32.2  : BOOL;
	O_LOADER_RS4_STOP AT %QX32.4  : BOOL;
	O_LOADER_RS4_PAUSE AT %QX32.5  : BOOL;
	O_LOADER_RS4_CONTINUE AT %QX32.6  : BOOL;
	O_LOADER_RS4_RESET AT %QX32.7  : BOOL;	
	
	O_LOADER_RS4_SETMOTORON AT %QX33.0  : BOOL;
	O_LOADER_RS4_SETMOTOROFF AT %QX33.1  : BOOL;
	O_LOADER_RS4_HOME AT %QX33.2  : BOOL;

I_LOADER_RS4_GRIPPER_CLOSE_1 AT %I* : BOOL;
I_LOADER_RS4_GRIPPER_CLOSE_2 AT %I* : BOOL;
I_LOADER_RS4_GRIPPER_CLOSE_3 AT %I* : BOOL;
I_LOADER_RS4_GRIPPER_CLOSE_4 AT %I* : BOOL;
I_LOADER_RS4_GRIPPER_OPEN_1 AT %I* : BOOL;
I_LOADER_RS4_GRIPPER_OPEN_2 AT %I* : BOOL;
I_LOADER_RS4_GRIPPER_OPEN_3 AT %I* : BOOL;
I_LOADER_RS4_GRIPPER_OPEN_4 AT %I* : BOOL;
I_LOADER_RS4_GRIPPER_EXT_DOWN_1 AT %I* : BOOL;
I_LOADER_RS4_GRIPPER_EXT_DOWN_2 AT %I* : BOOL;
I_LOADER_RS4_GRIPPER_EXT_DOWN_3 AT %I* : BOOL;
I_LOADER_RS4_GRIPPER_EXT_DOWN_4 AT %I* : BOOL;
I_LOADER_RS4_GRIPPER_EXT_UP_1 AT %I* : BOOL;
I_LOADER_RS4_GRIPPER_EXT_UP_2 AT %I* : BOOL;
I_LOADER_RS4_GRIPPER_EXT_UP_3 AT %I* : BOOL;
I_LOADER_RS4_GRIPPER_EXT_UP_4 AT %I* : BOOL;

O_LOADER_RS4_GRIPPER_CLOSE_1 AT %Q* : BOOL;
O_LOADER_RS4_GRIPPER_CLOSE_2 AT %Q* : BOOL;
O_LOADER_RS4_GRIPPER_CLOSE_3 AT %Q* : BOOL;
O_LOADER_RS4_GRIPPER_CLOSE_4 AT %Q* : BOOL;
O_LOADER_RS4_GRIPPER_OPEN_1 AT %Q* : BOOL;
O_LOADER_RS4_GRIPPER_OPEN_2 AT %Q* : BOOL;
O_LOADER_RS4_GRIPPER_OPEN_3 AT %Q* : BOOL;
O_LOADER_RS4_GRIPPER_OPEN_4 AT %Q* : BOOL;
O_LOADER_RS4_GRIPPER_EXT_DOWN_1 AT %Q* : BOOL;
O_LOADER_RS4_GRIPPER_EXT_DOWN_2 AT %Q* : BOOL;
O_LOADER_RS4_GRIPPER_EXT_DOWN_3 AT %Q* : BOOL;
O_LOADER_RS4_GRIPPER_EXT_DOWN_4 AT %Q* : BOOL;
O_LOADER_RS4_GRIPPER_EXT_UP_1 AT %Q* : BOOL;
O_LOADER_RS4_GRIPPER_EXT_UP_2 AT %Q* : BOOL;
O_LOADER_RS4_GRIPPER_EXT_UP_3 AT %Q* : BOOL;
O_LOADER_RS4_GRIPPER_EXT_UP_4 AT %Q* : BOOL;

IX_LOADER_RS4_GRIPPER_1 AT %IX36.0 : BOOL;
IX_LOADER_RS4_GRIPPER_2 AT %IX36.1 : BOOL;
IX_LOADER_RS4_GRIPPER_3 AT %IX36.2 : BOOL;
IX_LOADER_RS4_GRIPPER_4 AT %IX36.3 : BOOL;

IX_LOADER_RS4_GRIPPER_EXT_1 AT %IX36.4 : BOOL;
IX_LOADER_RS4_GRIPPER_EXT_2 AT %IX36.5 : BOOL;
IX_LOADER_RS4_GRIPPER_EXT_3 AT %IX36.6 : BOOL;
IX_LOADER_RS4_GRIPPER_EXT_4 AT %IX36.7 : BOOL;

(*
OX_LOADER_RS4_GRIPPER_1 AT %QX69.0 : BOOL;
OX_LOADER_RS4_GRIPPER_2 AT %QX69.1 : BOOL;
OX_LOADER_RS4_GRIPPER_3 AT %QX69.2 : BOOL;
OX_LOADER_RS4_GRIPPER_4 AT %QX69.3 : BOOL;

OX_LOADER_RS4_GRIPPER_EXT_1 AT %QX69.4 : BOOL;
OX_LOADER_RS4_GRIPPER_EXT_2 AT %QX69.5 : BOOL;
OX_LOADER_RS4_GRIPPER_EXT_3 AT %QX69.6 : BOOL;
OX_LOADER_RS4_GRIPPER_EXT_4 AT %QX69.7 : BOOL;
*)

IX_LOADER_RS4_HOME AT %I* : BOOL;
IX_LOADER_RS4_RUNNING AT %I* : BOOL;
IX_LOADER_RS4_PICKUP_1 AT %I* : BOOL;
IX_LOADER_RS4_PICKUP_2 AT %I* : BOOL;
IX_LOADER_RS4_PICKUP_3 AT %I* : BOOL;
IX_LOADER_RS4_PICKUP_4 AT %I* : BOOL;
IX_LOADER_RS4_PLACING_1 AT %I* : BOOL;
IX_LOADER_RS4_PLACING_2 AT %I* : BOOL;
IX_LOADER_RS4_PLACING_3 AT %I* : BOOL;
IX_LOADER_RS4_PLACING_4 AT %I* : BOOL;

IX_LOADER_RS4_FINISH AT %I* : BOOL;
I_LOADER_RS4_HANG :BOOL;
I_LOADER_RS4_END_CARRIER :BOOL;
I_LOADER_RS4_ENABLE :BOOL;
I_LOADER_RS4_DISABLE :BOOL;

END_VAR

// ---- GVLs/LOADER_VAR.TcGVL
{attribute 'qualified_only'}
VAR_GLOBAL
I_LOADER_CLAMPING_ON_1 AT %I* : BOOL;
I_LOADER_CLAMPING_ON_2 AT %I* : BOOL;
I_LOADER_CLAMPING_ON_3 AT %I* : BOOL;
I_LOADER_CLAMPING_ON_4 AT %I* : BOOL;
I_LOADER_CLAMPING_OFF_1 AT %I* : BOOL;
I_LOADER_CLAMPING_OFF_2 AT %I* : BOOL;
I_LOADER_CLAMPING_OFF_3 AT %I* : BOOL;
I_LOADER_CLAMPING_OFF_4 AT %I* : BOOL;

I_C8_FRONT_LIMIT AT %I* : BOOL;
I_C8_REAR_LIMIT AT %I* : BOOL;
I_ENABLE_SWITCH AT %I* : BOOL;
I_DISABLE_SWITCH AT %I* : BOOL;
I_EMERGENCY_SWITCH AT %I* : BOOL;
I_SAFETY_CURTAIN_1 AT %I* : BOOL;
I_SAFETY_CURTAIN_2 AT %I* : BOOL;
I_BUYOFF_RACK_1 AT %I* : BOOL;
I_BUYOFF_RACK_2 AT %I* : BOOL;
I_BUYOFF_RACK_3 AT %I* : BOOL;
I_BUYOFF_RACK_4 AT %I* : BOOL;
I_BUYOFF_RACK_5 AT %I* : BOOL;
I_BUYOFF_RACK_6 AT %I* : BOOL;
I_BUYOFF_RACK_7 AT %I* : BOOL;
I_BUYOFF_RACK_8 AT %I* : BOOL;
I_BUYOFF_RACK_9 AT %I* : BOOL;
I_BUYOFF_RACK_10 AT %I* : BOOL;
I_BUYOFF_RACK_11 AT %I* : BOOL;
I_BUYOFF_RACK_12 AT %I* : BOOL;
I_BUYOFF_RACK_13 AT %I* : BOOL;
I_BUYOFF_RACK_14 AT %I* : BOOL;
I_BUYOFF_RACK_15 AT %I* : BOOL;
I_BUYOFF_RACK_16 AT %I* : BOOL;
I_BUYOFF_RACK_17 AT %I* : BOOL;
I_BUYOFF_RACK_18 AT %I* : BOOL;
I_BUYOFF_RACK_19 AT %I* : BOOL;
I_BUYOFF_RACK_20 AT %I* : BOOL;
I_BUYOFF_RACK_21 AT %I* : BOOL;
I_BUYOFF_RACK_22 AT %I* : BOOL;
I_BUYOFF_RACK_23 AT %I* : BOOL;
I_BUYOFF_RACK_24 AT %I* : BOOL;
I_C8_GRIPPER_ON AT %I* : BOOL;
I_C8_GRIPPER_OFF AT %I* : BOOL;
I_SAFETY_FENCE_OPEN_1 AT %I* : BOOL;
I_SAFETY_FENCE_OPEN_2 AT %I* : BOOL;
I_SAFETY_FENCE_OPEN_3 AT %I* : BOOL;
I_SAFETY_FENCE_OPEN_4 AT %I* : BOOL;
I_SAFETY_FENCE_OPEN_5 AT %I* : BOOL;
I_SAFETY_FENCE_OPEN_6 AT %I* : BOOL;
I_SAFETY_FENCE_OPEN_7 AT %I* : BOOL;
I_SAFETY_FENCE_OPEN_8 AT %I* : BOOL;
I_SAFETY_FENCE_OPEN_9 AT %I* : BOOL;
I_SAFETY_FENCE_OPEN_10 AT %I* : BOOL;
I_SAFETY_FENCE_OPEN_11 AT %I* : BOOL;
I_SAFETY_FENCE_OPEN_12 AT %I* : BOOL;
I_SAFETY_FENCE_LOCK_ON_1 AT %I* : BOOL;
I_SAFETY_FENCE_LOCK_ON_2 AT %I* : BOOL;
I_SAFETY_FENCE_LOCK_ON_3 AT %I* : BOOL;
I_SAFETY_FENCE_LOCK_ON_4 AT %I* : BOOL;
I_SAFETY_FENCE_LOCK_ON_5 AT %I* : BOOL;
I_SAFETY_FENCE_LOCK_ON_6 AT %I* : BOOL;
I_SAFETY_FENCE_LOCK_ON_7 AT %I* : BOOL;
I_SAFETY_FENCE_LOCK_ON_8 AT %I* : BOOL;
I_SAFETY_FENCE_LOCK_ON_9 AT %I* : BOOL;
I_SAFETY_FENCE_LOCK_ON_10 AT %I* : BOOL;
I_SAFETY_FENCE_LOCK_ON_11 AT %I* : BOOL;
I_SAFETY_FENCE_LOCK_ON_12 AT %I* : BOOL;
I_SAFETY_FENCE_LOCK_OFF_1 AT %I* : BOOL;
I_SAFETY_FENCE_LOCK_OFF_2 AT %I* : BOOL;
I_SAFETY_FENCE_LOCK_OFF_3 AT %I* : BOOL;
I_SAFETY_FENCE_LOCK_OFF_4 AT %I* : BOOL;
I_SAFETY_FENCE_LOCK_OFF_5 AT %I* : BOOL;
I_SAFETY_FENCE_LOCK_OFF_6 AT %I* : BOOL;
I_SAFETY_FENCE_LOCK_OFF_7 AT %I* : BOOL;
I_SAFETY_FENCE_LOCK_OFF_8 AT %I* : BOOL;
I_SAFETY_FENCE_LOCK_OFF_9 AT %I* : BOOL;
I_SAFETY_FENCE_LOCK_OFF_10 AT %I* : BOOL;
I_SAFETY_FENCE_LOCK_OFF_11 AT %I* : BOOL;
I_SAFETY_FENCE_LOCK_OFF_12 AT %I* : BOOL;
I_TESTER_ENABLE_1 AT %I* : BOOL;
I_TESTER_ENABLE_2 AT %I* : BOOL;
I_TESTER_ENABLE_3 AT %I* : BOOL;
I_TESTER_ENABLE_4 AT %I* : BOOL;
I_TESTER_ENABLE_5 AT %I* : BOOL;
I_TESTER_ENABLE_6 AT %I* : BOOL;
I_TESTER_ENABLE_7 AT %I* : BOOL;
I_TESTER_ENABLE_8 AT %I* : BOOL;
I_TESTER_ENABLE_9 AT %I* : BOOL;
I_TESTER_ENABLE_10 AT %I* : BOOL;
I_TESTER_ENABLE_11 AT %I* : BOOL;
I_TESTER_ENABLE_12 AT %I* : BOOL;
I_TESTER_DISABLE_1 AT %I* : BOOL;
I_TESTER_DISABLE_2 AT %I* : BOOL;
I_TESTER_DISABLE_3 AT %I* : BOOL;
I_TESTER_DISABLE_4 AT %I* : BOOL;
I_TESTER_DISABLE_5 AT %I* : BOOL;
I_TESTER_DISABLE_6 AT %I* : BOOL;
I_TESTER_DISABLE_7 AT %I* : BOOL;
I_TESTER_DISABLE_8 AT %I* : BOOL;
I_TESTER_DISABLE_9 AT %I* : BOOL;
I_TESTER_DISABLE_10 AT %I* : BOOL;
I_TESTER_DISABLE_11 AT %I* : BOOL;
I_TESTER_DISABLE_12 AT %I* : BOOL;
I_TESTER_EMERGENCY_1 AT %I* : BOOL;
I_TESTER_EMERGENCY_2 AT %I* : BOOL;
I_TESTER_EMERGENCY_3 AT %I* : BOOL;
I_TESTER_EMERGENCY_4 AT %I* : BOOL;
I_TESTER_EMERGENCY_5 AT %I* : BOOL;
I_TESTER_EMERGENCY_6 AT %I* : BOOL;
I_TESTER_EMERGENCY_7 AT %I* : BOOL;
I_TESTER_EMERGENCY_8 AT %I* : BOOL;
I_TESTER_EMERGENCY_9 AT %I* : BOOL;
I_TESTER_EMERGENCY_10 AT %I* : BOOL;
I_TESTER_EMERGENCY_11 AT %I* : BOOL;
I_TESTER_EMERGENCY_12 AT %I* : BOOL;
I_BUFFER_CARRIER_DETECT_1 AT %I* : BOOL;
I_BUFFER_CARRIER_DETECT_2 AT %I* : BOOL;
I_INPUT_CARTESSIAN_HOME AT %I* : BOOL;
I_INPUT_CARTESSIAN_RUNNING AT %I* : BOOL;
I_INPUT_CARTESSIAN_FINISH AT %I* : BOOL;


O_LOADER_CLAMPING_ON_1 AT %Q* : BOOL;
O_LOADER_CLAMPING_ON_2 AT %Q* : BOOL;
O_LOADER_CLAMPING_ON_3 AT %Q* : BOOL;
O_LOADER_CLAMPING_ON_4 AT %Q* : BOOL;
O_LOADER_CLAMPING_OFF_1 AT %Q* : BOOL;
O_LOADER_CLAMPING_OFF_2 AT %Q* : BOOL;
O_LOADER_CLAMPING_OFF_3 AT %Q* : BOOL;
O_LOADER_CLAMPING_OFF_4 AT %Q* : BOOL;
O_C8_GRIPPER_ON AT %Q* : BOOL;
O_C8_GRIPPER_OFF AT %Q* : BOOL;
O_SAFETY_FENCE_LOCK_ON_1 AT %Q* : BOOL;
O_SAFETY_FENCE_LOCK_ON_2 AT %Q* : BOOL;
O_SAFETY_FENCE_LOCK_ON_3 AT %Q* : BOOL;
O_SAFETY_FENCE_LOCK_ON_4 AT %Q* : BOOL;
O_SAFETY_FENCE_LOCK_ON_5 AT %Q* : BOOL;
O_SAFETY_FENCE_LOCK_ON_6 AT %Q* : BOOL;
O_SAFETY_FENCE_LOCK_ON_7 AT %Q* : BOOL;
O_SAFETY_FENCE_LOCK_ON_8 AT %Q* : BOOL;
O_SAFETY_FENCE_LOCK_ON_9 AT %Q* : BOOL;
O_SAFETY_FENCE_LOCK_ON_10 AT %Q* : BOOL;
O_SAFETY_FENCE_LOCK_ON_11 AT %Q* : BOOL;
O_SAFETY_FENCE_LOCK_ON_12 AT %Q* : BOOL;
O_TESTER_TOWER_LAMP_RED_1 AT %Q* : BOOL;
O_TESTER_TOWER_LAMP_RED_2 AT %Q* : BOOL;
O_TESTER_TOWER_LAMP_RED_3 AT %Q* : BOOL;
O_TESTER_TOWER_LAMP_RED_4 AT %Q* : BOOL;
O_TESTER_TOWER_LAMP_RED_5 AT %Q* : BOOL;
O_TESTER_TOWER_LAMP_RED_6 AT %Q* : BOOL;
O_TESTER_TOWER_LAMP_RED_7 AT %Q* : BOOL;
O_TESTER_TOWER_LAMP_RED_8 AT %Q* : BOOL;
O_TESTER_TOWER_LAMP_RED_9 AT %Q* : BOOL;
O_TESTER_TOWER_LAMP_RED_10 AT %Q* : BOOL;
O_TESTER_TOWER_LAMP_RED_11 AT %Q* : BOOL;
O_TESTER_TOWER_LAMP_RED_12 AT %Q* : BOOL;
O_TESTER_TOWER_LAMP_YELLOW_1 AT %Q* : BOOL;
O_TESTER_TOWER_LAMP_YELLOW_2 AT %Q* : BOOL;
O_TESTER_TOWER_LAMP_YELLOW_3 AT %Q* : BOOL;
O_TESTER_TOWER_LAMP_YELLOW_4 AT %Q* : BOOL;
O_TESTER_TOWER_LAMP_YELLOW_5 AT %Q* : BOOL;
O_TESTER_TOWER_LAMP_YELLOW_6 AT %Q* : BOOL;
O_TESTER_TOWER_LAMP_YELLOW_7 AT %Q* : BOOL;
O_TESTER_TOWER_LAMP_YELLOW_8 AT %Q* : BOOL;
O_TESTER_TOWER_LAMP_YELLOW_9 AT %Q* : BOOL;
O_TESTER_TOWER_LAMP_YELLOW_10 AT %Q* : BOOL;
O_TESTER_TOWER_LAMP_YELLOW_11 AT %Q* : BOOL;
O_TESTER_TOWER_LAMP_YELLOW_12 AT %Q* : BOOL;
O_TESTER_TOWER_LAMP_GREEN_1 AT %Q* : BOOL;
O_TESTER_TOWER_LAMP_GREEN_2 AT %Q* : BOOL;
O_TESTER_TOWER_LAMP_GREEN_3 AT %Q* : BOOL;
O_TESTER_TOWER_LAMP_GREEN_4 AT %Q* : BOOL;
O_TESTER_TOWER_LAMP_GREEN_5 AT %Q* : BOOL;
O_TESTER_TOWER_LAMP_GREEN_6 AT %Q* : BOOL;
O_TESTER_TOWER_LAMP_GREEN_7 AT %Q* : BOOL;
O_TESTER_TOWER_LAMP_GREEN_8 AT %Q* : BOOL;
O_TESTER_TOWER_LAMP_GREEN_9 AT %Q* : BOOL;
O_TESTER_TOWER_LAMP_GREEN_10 AT %Q* : BOOL;
O_TESTER_TOWER_LAMP_GREEN_11 AT %Q* : BOOL;
O_TESTER_TOWER_LAMP_GREEN_12 AT %Q* : BOOL;
O_TESTER_CHILLER_ON_1 AT %Q* : BOOL;
O_TESTER_CHILLER_ON_2 AT %Q* : BOOL;
O_TESTER_CHILLER_ON_3 AT %Q* : BOOL;
O_TESTER_CHILLER_ON_4 AT %Q* : BOOL;
O_TESTER_CHILLER_ON_5 AT %Q* : BOOL;
O_TESTER_CHILLER_ON_6 AT %Q* : BOOL;
O_TESTER_CHILLER_ON_7 AT %Q* : BOOL;
O_TESTER_CHILLER_ON_8 AT %Q* : BOOL;
O_TESTER_CHILLER_ON_9 AT %Q* : BOOL;
O_TESTER_CHILLER_ON_10 AT %Q* : BOOL;
O_TESTER_CHILLER_ON_11 AT %Q* : BOOL;
O_TESTER_CHILLER_ON_12 AT %Q* : BOOL;
O_TESTER_CHILLER_OFF_1 AT %Q* : BOOL;
O_TESTER_CHILLER_OFF_2 AT %Q* : BOOL;
O_TESTER_CHILLER_OFF_3 AT %Q* : BOOL;
O_TESTER_CHILLER_OFF_4 AT %Q* : BOOL;
O_TESTER_CHILLER_OFF_5 AT %Q* : BOOL;
O_TESTER_CHILLER_OFF_6 AT %Q* : BOOL;
O_TESTER_CHILLER_OFF_7 AT %Q* : BOOL;
O_TESTER_CHILLER_OFF_8 AT %Q* : BOOL;
O_TESTER_CHILLER_OFF_9 AT %Q* : BOOL;
O_TESTER_CHILLER_OFF_10 AT %Q* : BOOL;
O_TESTER_CHILLER_OFF_11 AT %Q* : BOOL;
O_TESTER_CHILLER_OFF_12 AT %Q* : BOOL;
O_TESTER_POWER_ON_1 AT %Q* : BOOL;
O_TESTER_POWER_ON_2 AT %Q* : BOOL;
O_TESTER_POWER_ON_3 AT %Q* : BOOL;
O_TESTER_POWER_ON_4 AT %Q* : BOOL;
O_TESTER_POWER_ON_5 AT %Q* : BOOL;
O_TESTER_POWER_ON_6 AT %Q* : BOOL;
O_TESTER_POWER_ON_7 AT %Q* : BOOL;
O_TESTER_POWER_ON_8 AT %Q* : BOOL;
O_TESTER_POWER_ON_9 AT %Q* : BOOL;
O_TESTER_POWER_ON_10 AT %Q* : BOOL;
O_TESTER_POWER_ON_11 AT %Q* : BOOL;
O_TESTER_POWER_ON_12 AT %Q* : BOOL;
O_TESTER_PC_SWITCH_ON_1 AT %Q* : BOOL;
O_TESTER_PC_SWITCH_ON_2 AT %Q* : BOOL;
O_TESTER_PC_SWITCH_ON_3 AT %Q* : BOOL;
O_TESTER_PC_SWITCH_ON_4 AT %Q* : BOOL;
O_TESTER_PC_SWITCH_ON_5 AT %Q* : BOOL;
O_TESTER_PC_SWITCH_ON_6 AT %Q* : BOOL;
O_TESTER_PC_SWITCH_ON_7 AT %Q* : BOOL;
O_TESTER_PC_SWITCH_ON_8 AT %Q* : BOOL;
O_TESTER_PC_SWITCH_ON_9 AT %Q* : BOOL;
O_TESTER_PC_SWITCH_ON_10 AT %Q* : BOOL;
O_TESTER_PC_SWITCH_ON_11 AT %Q* : BOOL;
O_TESTER_PC_SWITCH_ON_12 AT %Q* : BOOL;
O_TESTER_START_1 AT %Q* : BOOL;
O_TESTER_START_2 AT %Q* : BOOL;
O_TESTER_START_3 AT %Q* : BOOL;
O_TESTER_START_4 AT %Q* : BOOL;
O_TESTER_START_5 AT %Q* : BOOL;
O_TESTER_START_6 AT %Q* : BOOL;
O_TESTER_START_7 AT %Q* : BOOL;
O_TESTER_START_8 AT %Q* : BOOL;
O_TESTER_START_9 AT %Q* : BOOL;
O_TESTER_START_10 AT %Q* : BOOL;
O_TESTER_START_11 AT %Q* : BOOL;
O_TESTER_START_12 AT %Q* : BOOL;
O_TESTER_STOP_1 AT %Q* : BOOL;
O_TESTER_STOP_2 AT %Q* : BOOL;
O_TESTER_STOP_3 AT %Q* : BOOL;
O_TESTER_STOP_4 AT %Q* : BOOL;
O_TESTER_STOP_5 AT %Q* : BOOL;
O_TESTER_STOP_6 AT %Q* : BOOL;
O_TESTER_STOP_7 AT %Q* : BOOL;
O_TESTER_STOP_8 AT %Q* : BOOL;
O_TESTER_STOP_9 AT %Q* : BOOL;
O_TESTER_STOP_10 AT %Q* : BOOL;
O_TESTER_STOP_11 AT %Q* : BOOL;
O_TESTER_STOP_12 AT %Q* : BOOL;

END_VAR

// ---- GVLs/SORTER_RS4_VAR.TcGVL
{attribute 'qualified_only'}
VAR_GLOBAL

SORTER_RS4_INPUT AT %IB64 : BYTE;  
SORTER_RS4_INPUT_1 AT %IB65 : BYTE; 
SORTER_RS4_INPUT_2 AT %IB66 : BYTE;  
SORTER_RS4_INPUT_3 AT %IB67 : BYTE; 
SORTER_RS4_INPUT_4 AT %IB68 : BYTE; 
SORTER_RS4_INPUT_5 AT %IB69 : BYTE; 
SORTER_RS4_INPUT_6 AT %IB70 : BYTE; 

SORTER_RS4_OUTPUT AT %QB64 : BYTE; 
SORTER_RS4_OUTPUT_1 AT %QB65 : BYTE; 
SORTER_RS4_POS_TAKEUP_1 AT %QB66 : BYTE:=1; 
SORTER_RS4_POS_TAKEUP_2 AT %QB67 : BYTE:=2;
SORTER_RS4_POS_TAKEUP_3 AT %QB68 : BYTE:=3; 
SORTER_RS4_POS_TAKEUP_4 AT %QB69 : BYTE:=4;
SORTER_RS4_POS_PLACING_1 AT %QB70 : BYTE:=1; 
SORTER_RS4_POS_PLACING_2 AT %QB71 : BYTE:=5;
SORTER_RS4_POS_PLACING_3 AT %QB72 : BYTE:=9; 
SORTER_RS4_POS_PLACING_4 AT %QB73 : BYTE:=9; 
SORTER_RS4_OUTPUT_10 AT %QB74 : BYTE;

I_SORTER_RS4_READY  AT %IX64.0 :BOOL;
I_SORTER_RS4_RUNNING  AT %IX64.1 :BOOL;
I_SORTER_RS4_PAUSED  AT %IX64.2 :BOOL;
I_SORTER_RS4_ERROR  AT %IX64.3 :BOOL;
I_SORTER_RS4_ESTOPON  AT %IX64.4 :BOOL;
I_SORTER_RS46_SAFEGUARDON  AT %IX64.5 :BOOL;
I_SORTER_RS4_SERROR  AT %IX64.6 :BOOL;
I_SORTER_RS4_WARNING  AT %IX64.7 :BOOL;

I_SORTER_RS4_MOTORON  AT %IX65.0 :BOOL;
I_SORTER_RS4_ATHOME  AT %IX65.1 :BOOL;
I_SORTER_RS4_AUTOMODE  AT %IX65.5 :BOOL;

IX_SORTER_RS4_GRIPPER_1 AT %IX66.0 : BOOL;
IX_SORTER_RS4_GRIPPER_2 AT %IX66.1 : BOOL;
IX_SORTER_RS4_GRIPPER_3 AT %IX66.2 : BOOL;
IX_SORTER_RS4_GRIPPER_4 AT %IX66.3 : BOOL;

IX_SORTER_RS4_GRIPPER_EXT_1 AT %IX66.4 : BOOL;
IX_SORTER_RS4_GRIPPER_EXT_2 AT %IX66.5 : BOOL;
IX_SORTER_RS4_GRIPPER_EXT_3 AT %IX66.6 : BOOL;
IX_SORTER_RS4_GRIPPER_EXT_4 AT %IX66.7 : BOOL;

I_SORTER_RS4_END_CYCLE  AT %IX67.0 :BOOL;
//I_SORTER_RS4_END_CARRIER  AT %IX69.1 :BOOL;
I_SORTER_RS4_READY_TAKEUP  AT %IX67.2 :BOOL;//CYCLE RUNNING INDICATOR
I_SORTER_RS4_START_TAKEUP  AT %IX67.3 :BOOL;
I_SORTER_RS4_READY_PLACING  AT %IX67.4 :BOOL;
I_SORTER_RS4_START_PLACING  AT %IX67.5 :BOOL;
	
	O_SORTER_RS4_START AT %QX64.0  : BOOL;	
	O_SORTER_RS4_SELECT_FUKUDA_A AT %QX64.1  : BOOL;
	O_SORTER_RS4_SELECT_FUKUDA_B AT %QX64.2  : BOOL;
	O_SORTER_RS4_STOP AT %QX64.4  : BOOL;
	O_SORTER_RS4_PAUSE AT %QX64.5  : BOOL;
	O_SORTER_RS4_CONTINUE AT %QX64.6  : BOOL;
	O_SORTER_RS4_RESET AT %QX64.7  : BOOL;	
	
	O_SORTER_RS4_SETMOTORON AT %QX65.0  : BOOL;
	O_SORTER_RS4_SETMOTOROFF AT %QX65.1  : BOOL;
	O_SORTER_RS4_HOME AT %QX65.2  : BOOL;

I_SORTER_RS4_GRIPPER_CLOSE_1 AT %I* : BOOL;
I_SORTER_RS4_GRIPPER_CLOSE_2 AT %I* : BOOL;
I_SORTER_RS4_GRIPPER_CLOSE_3 AT %I* : BOOL;
I_SORTER_RS4_GRIPPER_CLOSE_4 AT %I* : BOOL;
I_SORTER_RS4_GRIPPER_OPEN_1 AT %I* : BOOL;
I_SORTER_RS4_GRIPPER_OPEN_2 AT %I* : BOOL;
I_SORTER_RS4_GRIPPER_OPEN_3 AT %I* : BOOL;
I_SORTER_RS4_GRIPPER_OPEN_4 AT %I* : BOOL;
I_SORTER_RS4_GRIPPER_EXT_DOWN_1 AT %I* : BOOL;
I_SORTER_RS4_GRIPPER_EXT_DOWN_2 AT %I* : BOOL;
I_SORTER_RS4_GRIPPER_EXT_DOWN_3 AT %I* : BOOL;
I_SORTER_RS4_GRIPPER_EXT_DOWN_4 AT %I* : BOOL;
I_SORTER_RS4_GRIPPER_EXT_UP_1 AT %I* : BOOL;
I_SORTER_RS4_GRIPPER_EXT_UP_2 AT %I* : BOOL;
I_SORTER_RS4_GRIPPER_EXT_UP_3 AT %I* : BOOL;
I_SORTER_RS4_GRIPPER_EXT_UP_4 AT %I* : BOOL;

O_SORTER_RS4_GRIPPER_CLOSE_1 AT %Q* : BOOL;
O_SORTER_RS4_GRIPPER_CLOSE_2 AT %Q* : BOOL;
O_SORTER_RS4_GRIPPER_CLOSE_3 AT %Q* : BOOL;
O_SORTER_RS4_GRIPPER_CLOSE_4 AT %Q* : BOOL;
O_SORTER_RS4_GRIPPER_OPEN_1 AT %Q* : BOOL;
O_SORTER_RS4_GRIPPER_OPEN_2 AT %Q* : BOOL;
O_SORTER_RS4_GRIPPER_OPEN_3 AT %Q* : BOOL;
O_SORTER_RS4_GRIPPER_OPEN_4 AT %Q* : BOOL;
O_SORTER_RS4_GRIPPER_EXT_DOWN_1 AT %Q* : BOOL;
O_SORTER_RS4_GRIPPER_EXT_DOWN_2 AT %Q* : BOOL;
O_SORTER_RS4_GRIPPER_EXT_DOWN_3 AT %Q* : BOOL;
O_SORTER_RS4_GRIPPER_EXT_DOWN_4 AT %Q* : BOOL;
O_SORTER_RS4_GRIPPER_EXT_UP_1 AT %Q* : BOOL;
O_SORTER_RS4_GRIPPER_EXT_UP_2 AT %Q* : BOOL;
O_SORTER_RS4_GRIPPER_EXT_UP_3 AT %Q* : BOOL;
O_SORTER_RS4_GRIPPER_EXT_UP_4 AT %Q* : BOOL;

IX_SORTER_RS4_HOME AT %I* : BOOL;
IX_SORTER_RS4_RUNNING AT %I* : BOOL;
IX_SORTER_RS4_PICKUP_1 AT %I* : BOOL;
IX_SORTER_RS4_PICKUP_2 AT %I* : BOOL;
IX_SORTER_RS4_PICKUP_3 AT %I* : BOOL;
IX_SORTER_RS4_PICKUP_4 AT %I* : BOOL;
IX_SORTER_RS4_PLACING_1 AT %I* : BOOL;
IX_SORTER_RS4_PLACING_2 AT %I* : BOOL;
IX_SORTER_RS4_PLACING_3 AT %I* : BOOL;
IX_SORTER_RS4_PLACING_4 AT %I* : BOOL;

IX_SORTER_RS4_FINISH AT %I* : BOOL;
I_SORTER_RS4_HANG :BOOL;
I_SORTER_RS4_END_CARRIER :BOOL;
I_SORTER_RS4_ENABLE :BOOL; 
I_SORTER_RS4_DISABLE :BOOL;

END_VAR

// ---- GVLs/SORTER_VAR.TcGVL
{attribute 'qualified_only'}
VAR_GLOBAL
I_LOTBOX_CLAMP_ON_1 AT %I* : BOOL;
I_LOTBOX_CLAMP_ON_2 AT %I* : BOOL;
I_LOTBOX_CLAMP_ON_3 AT %I* : BOOL;
I_LOTBOX_CLAMP_ON_4 AT %I* : BOOL;
I_LOTBOX_CLAMP_OFF_1 AT %I* : BOOL;
I_LOTBOX_CLAMP_OFF_2 AT %I* : BOOL;
I_LOTBOX_CLAMP_OFF_3 AT %I* : BOOL;
I_LOTBOX_CLAMP_OFF_4 AT %I* : BOOL;
	
I_LOTBOX_DETECT_1 AT %I* : BOOL;//LOTBOX_LASER1_DETECT
I_LOTBOX_DETECT_2 AT %I* : BOOL;//LOTBOX_LASER2_DETECT
I_LOTBOX_DETECT_3 AT %I* : BOOL;//LOTBOX_LASER3_DETECT
I_LOTBOX_DETECT_4 AT %I* : BOOL;//LOTBOX_LASER4_DETECT

I_VACUUM_ON AT %I* : BOOL;
I_VACUUM_OFF AT %I* : BOOL;

I_LASER_TRANSFER_AT_FRONT_A AT %I* : BOOL;
I_LASER_TRANSFER_AT_BACK_A AT %I* : BOOL;
I_LASER_TRANSFER_AT_FRONT_B AT %I* : BOOL;
I_LASER_TRANSFER_AT_BACK_B AT %I* : BOOL;
I_LASER_TRANSFER_A_PICK_DONE : BOOL;
I_LASER_TRANSFER_B_PICK_DONE : BOOL;
I_LASER_TRANSFER_AT_A : BOOL;
I_LASER_TRANSFER_AT_B : BOOL;

//I_LOTEND :BOOL :=FALSE;
I_FUNC_CALLED:BOOL:=FALSE;
I_LOADING_DONE : BOOL;
I_LOADING_FAILED: BOOL;
I_LOADING_ALARM: INT;
I_CURRENT_TRANSACTION : T_CURRENT_TRANSACTION ; 
I_CARTESSIAN_GRIPPER_ON AT %I* : BOOL;
I_CARTESSIAN_GRIPPER_OFF AT %I* : BOOL;
I_FUNCTION_NAME :STRING [255];
I_CASE : INT:=0;
I_LASER_RUNNING:BOOL :=FALSE;

O_LOTBOX_CLAMP_ON_1 AT %Q* : BOOL;
O_LOTBOX_CLAMP_ON_2 AT %Q* : BOOL;
O_LOTBOX_CLAMP_ON_3 AT %Q* : BOOL;
O_LOTBOX_CLAMP_ON_4 AT %Q* : BOOL;
O_LOTBOX_CLAMP_OFF_1 AT %Q* : BOOL;
O_LOTBOX_CLAMP_OFF_2 AT %Q* : BOOL;
O_LOTBOX_CLAMP_OFF_3 AT %Q* : BOOL;
O_LOTBOX_CLAMP_OFF_4 AT %Q* : BOOL;

O_VACUUM_ON AT %Q* : BOOL;
O_VACUUM_OFF AT %Q* : BOOL;
O_CARTESSIAN_GRIPPER_ON AT %Q* : BOOL;
O_CARTESSIAN_GRIPPER_OFF AT %Q* : BOOL;
O_TOWER_LAMP_RED AT %Q* : BOOL;
O_TOWER_LAMP_YELLOW AT %Q* : BOOL;
O_TOWER_LAMP_GREEN AT %Q* : BOOL;
O_TOWER_LAMP_BUZZER AT %Q* : BOOL;
O_WARNING_LIGHT AT %Q* : BOOL;
O_LOT_BOX_INDICATOR_1  AT %Q* : BOOL;
O_LOT_BOX_INDICATOR_2 AT %Q* : BOOL;
O_LOT_BOX_INDICATOR_3 AT %Q* : BOOL;
O_LOT_BOX_INDICATOR_4 AT %Q* : BOOL;

AXIS_COMPLETE: BOOL;
JIG_LASER_PRESENCE: BOOL;
LOTBOX_READY_1: BOOL;

DataWordInput1 AT %IB232 : ARRAY [0..15] OF WORD; 
DataWordInput2 AT %IB264 : ARRAY [16..31] OF WORD;
DataWordInput3 AT %IB296 : ARRAY [32..47] OF WORD; 
DataWordInput4 AT %IB328 : ARRAY [48..56] OF WORD; 
DataWordOutput1 AT %QB232 : ARRAY [0..15] OF WORD; 
DataWordOutput2 AT %QB264 : ARRAY [16..31] OF WORD; 
DataWordOutput3 AT %QB296 : ARRAY [32..47] OF WORD; 
DataWordOutput4 AT %QB328 : ARRAY [48..56] OF WORD; 

O_NG_DATA_OUTPUT1 AT %Q* : BOOL;
O_NG_DATA_OUTPUT2 AT %Q* : BOOL;
O_NG_DATA_OUTPUT3 AT %Q* : BOOL;
O_NG_DATA_OUTPUT4 AT %Q* : BOOL;
O_NG_DATA_STOP AT %Q* : BOOL;
O_NG_DATA_RESET AT %Q* : BOOL;

I_NG_TRANSFER_AT_BACK AT %I* : BOOL;
I_NG_TRANSFER_AT_FRONT AT %I* : BOOL;

I_RETURN_DONE_A: BOOL;
I_RETURN_DONE_B: BOOL;
I_LOADING_DONE_A: BOOL;
I_LOADING_DONE_B: BOOL;
I_RETURN_ALARM: INT;
I_RETURN_FAILED: BOOL;
ACTIVE_ID: INT :=1;	
ACTIVE_PROGRAM: INT ;
ACTIVE_PROGRAM_CHANGE:BOOL;
	
I_LASER_HOME : BOOL;
O_LASER_HOME : BOOL;

STRAIGHTEN_START: BOOL;
STRAIGHTEN_PROCESS: BOOL;
STRAIGHTEN_DONE: BOOL;

LASER_HOME: BOOL;

O_STOPPER_TRANSFER_A AT %Q* : BOOL;
O_STOPPER_TRANSFER_B AT %Q* : BOOL;
I_STOPPER_TRANSFER_ON_A AT %Q* : BOOL;
I_STOPPER_TRANSFER_OFF_A AT %Q* : BOOL;
I_STOPPER_TRANSFER_ON_B AT %Q* : BOOL;
I_STOPPER_TRANSFER_OFF_B AT %Q* : BOOL;
O_RESET_CARTESSIAN: BOOL;
END_VAR

// ---- GVLs/TESTER_C8_VAR.TcGVL
{attribute 'qualified_only'}
VAR_GLOBAL
	
I_C8_GRIPPER_CLOSE AT %IX96.0 : BOOL;
I_C8_GRIPPER_OPEN AT %IX96.1 : BOOL;
I_C8_GBUFFER_1 AT %IX96.2 : BOOL;
I_C8_BUFFER_2 AT %IX96.3 : BOOL;

O_C8_GRIPPER_CLOSE AT %QX96.0 : BOOL;
O_C8_GRIPPER_OPEN AT %QX96.1 : BOOL;

C8_INPUT AT %IB96 :ARRAY [0..15]  OF WORD;
C8_OUTPUT AT %QB96 : BYTE;

(*
	I_C8_HOME AT %IX01.0 : BOOL;
	I_C8_PICKING_START AT %IX01.1  : BOOL;
	I_C8_PICKING_PROCESS AT %IX01.2  : BOOL;
	I_C8_PICKING_DONE  AT %IX01.3 :BOOL;
	I_C8_PLACING_START AT %IX01.4  : BOOL;
	I_C8_PLACING_PROCESS AT %IX01.5  : BOOL;
	I_C8_PLACING_DONE  AT %IX01.6 :BOOL;
	
	O_C8_HOME AT %QX102.0 : BOOL;
	O_C8_PICKING_START AT %QX102.1 : BOOL;
	O_C8_PICKING_STOP AT %QX102.2 : BOOL;
	O_C8_PLACING_START AT %QX102.3 : BOOL;
	O_C8_PLACING_STOP AT %QX102.4 : BOOL;
*)
END_VAR

// ---- POUs/MAIN.TcPOU
 PROGRAM MAIN

VAR

	EKE: BOOL; 
	STEP: INT :=1;
	
	TMR100: TON;
	stage: INT :=0;
	IC_CASE: INT :=0;
	
	START_STR: F_TRIG;
	START_G6: R_TRIG;
	I_RS4_PICKING_DONE: BOOL;
	START_STRAIGHTENER: R_TRIG;
	READY_1: BOOL;
	READY_2: BOOL;
	RR: BOOL;
	RX: R_TRIG;
	TRIG_IND2: R_TRIG;
END_VAR


//INPUT_CARTESSIAN(); 
INPUT_G6();
INDEXING();
INDEXING_2();
INPUT_PROG();
LOADER_RS4();
SORTER_RS4();
STRAIGHTENING_PROG_1();

(*
//EXECUTE_FUNCTION(INPUT_VAR.I_FUNCTION_NAME);

//LOAD_FUKUDA();
//MOVE STATION & JIG INDEX 


(************.::INDEXING 1 OPERATION::.***********) 
//LOADER_RS4_VAR.I_LOADER_RS4_READY_TAKEUP AND INPUT_G6_VAR.I_G6_READY_PLACING 
(*
IF INPUT_G6_VAR.I_G6_START_TAKEUP  THEN
	READY_1 :=TRUE;	
END_IF
IF LOADER_RS4_VAR.I_LOADER_RS4_START_PLACING  THEN
	READY_2 :=TRUE;
END_IF
*)

//START ROTATION INDEXING 1
READY_1 :=INPUT_G6_VAR.I_G6_START_TAKEUP;
READY_2 :=LOADER_RS4_VAR.I_LOADER_RS4_START_PLACING;
IF INDEXING_1_VAR.READY_STRAIGTHEN THEN
	READY_1 :=FALSE;	
	READY_2 :=FALSE;	
END_IF

IF READY_1 AND READY_2 AND INDEXING_1_VAR.I_INDEXING_1_ROTATION_DONE THEN//READY_PLACING THEN
	RR:=TRUE;
	RX(CLK:=RR);
	INDEXING_1_VAR.O_ROTATION_START:=RX.Q;
ELSE
	RR:=FALSE;
//RX(IN:=FALSE);
	RX(CLK:=FALSE);
END_IF


//START ROTATION INDEXING 2
IF SORTER_RS4_VAR.I_SORTER_RS4_END_CARRIER AND LOADER_RS4_VAR.I_LOADER_RS4_END_CARRIER THEN
	TRIG_IND2(CLK:=TRUE);
	INDEXING_2_VAR.O_ROTATION_START:=TRIG_IND2.Q;
	SORTER_RS4_VAR.I_SORTER_RS4_END_CARRIER:=FALSE;
	LOADER_RS4_VAR.I_LOADER_RS4_END_CARRIER:=FALSE;
	ELSE
	TRIG_IND2(CLK:=FALSE);
END_IF
*)
//CARTESSIAN INPUT
IF FLAG_VAR.ALLOW_EXECUTE_LOAD_FUKUDA THEN 
	IF INPUT_VAR.I_CASE=100 THEN
		INPUT_VAR.I_CASE:=0;
		IC_CASE:=0;	
		END_IF			
	LOAD_FUKUDA();
END_IF
IF FLAG_VAR.ALLOW_EXECUTE_RETURN_FUKUDA THEN 
	IF INPUT_VAR.I_CASE=100 THEN
		INPUT_VAR.I_CASE:=0;
		IC_CASE:=0;
	END_IF	
	RETURN_FUKUDA();	
END_IF

IF FLAG_VAR.ALLOW_EXECUTE_LOAD_LASER THEN 
	IF SORTER_VAR.I_CASE=100 THEN
		SORTER_VAR.I_CASE:=0;
		IC_CASE:=0;	
		END_IF			 
	LOAD_LASER();
END_IF
IF FLAG_VAR.ALLOW_EXECUTE_RETURN_LASER THEN 
	IF SORTER_VAR.I_CASE=100 THEN
		SORTER_VAR.I_CASE:=0;
		IC_CASE:=0;
	END_IF	
	RETURN_LASER();	
END_IF

IF FLAG_VAR.ALLOW_EXECUTE_LOAD_NG THEN 
	LOAD_NG();	
END_IF

IF FLAG_VAR.ALLOW_EXECUTE_RETURN_NG THEN 
	RETURN_NG();	
END_IF

END_PROGRAM

// ---- POUs/ROBOT/INPUT_G6.TcPOU
PROGRAM INPUT_G6
VAR
(*	
ROBOT_I_GRIPPER_1 AT %IX100.0 : BOOL;
	ROBOT_I_GRIPPER_2 AT %IX100.1 : BOOL;
	ROBOT_I_GRIPPER_3 AT %IX100.2 : BOOL;
	ROBOT_I_GRIPPER_4 AT %IX100.3 : BOOL;
	
	ROBOT_I_GRIPPER_EXT_1 AT %IX100.4 : BOOL;
	ROBOT_I_GRIPPER_EXT_2 AT %IX100.5 : BOOL;
	ROBOT_I_GRIPPER_EXT_3 AT %IX100.6 : BOOL;
	ROBOT_I_GRIPPER_EXT_4 AT %IX100.7 : BOOL;
	
	ROBOT_O_GRIPPER_1 AT %IX101.0 : BOOL;
	ROBOT_O_GRIPPER_2 AT %IX101.1 : BOOL;
	ROBOT_O_GRIPPER_3 AT %IX101.2 : BOOL;
	ROBOT_O_GRIPPER_4 AT %IX101.3 : BOOL;
		
	ROBOT_O_GRIPPER_EXT_1 AT %IX101.4 : BOOL;
	ROBOT_O_GRIPPER_EXT_2 AT %IX101.5 : BOOL;
	ROBOT_O_GRIPPER_EXT_3 AT %IX101.6 : BOOL;
	ROBOT_O_GRIPPER_EXT_4 AT %IX101.7 : BOOL;
	
	*)
	TMR11: TON;
	TMR12: TON;
	TMR10: TON;
	TMR8: TON;
	TMR9: TON;
	TMR7: TON;
	TMR3: TON;
	TP1: TP;
	TMR1: TON;
	START_ROBOT: TP;
	TP2: TP;
	O_G6_HANG: BOOL;
	I_G6_HANG: BOOL;
	TMR2: TON;
	GO_ROBOT: BOOL;
	TP3: TP;
	TMR4: TON;
	CNT_CYCLE: CTU;
	START_ROTATE: R_TRIG;
	IN: INT;
	TP_END_FUKUDA: TP;
	CNT_END_FUKUDA: CTU;
END_VAR

IF INPUT_G6_VAR.I_G6_ENABLE  THEN
//GRIPPING 
IF INPUT_G6_VAR.IX_G6_GRIPPER_1 THEN
	INPUT_G6_VAR.O_G6_GRIPPER_CLOSE_1:=TRUE;
	INPUT_G6_VAR.O_G6_GRIPPER_OPEN_1:=FALSE;
ELSE
	INPUT_G6_VAR.O_G6_GRIPPER_CLOSE_1:=FALSE;
	INPUT_G6_VAR.O_G6_GRIPPER_OPEN_1:=TRUE;
END_IF

IF INPUT_G6_VAR.IX_G6_GRIPPER_2 THEN
	INPUT_G6_VAR.O_G6_GRIPPER_CLOSE_2:=TRUE;
	INPUT_G6_VAR.O_G6_GRIPPER_OPEN_2:=FALSE;
ELSE
	INPUT_G6_VAR.O_G6_GRIPPER_CLOSE_2:=FALSE;
	INPUT_G6_VAR.O_G6_GRIPPER_OPEN_2:=TRUE;
END_IF 

IF INPUT_G6_VAR.IX_G6_GRIPPER_3 THEN
	INPUT_G6_VAR.O_G6_GRIPPER_CLOSE_3:=TRUE;
	INPUT_G6_VAR.O_G6_GRIPPER_OPEN_3:=FALSE;
ELSE
	INPUT_G6_VAR.O_G6_GRIPPER_CLOSE_3:=FALSE;
	INPUT_G6_VAR.O_G6_GRIPPER_OPEN_3:=TRUE;
END_IF

IF INPUT_G6_VAR.IX_G6_GRIPPER_4 THEN
	INPUT_G6_VAR.O_G6_GRIPPER_CLOSE_4:=TRUE;
	INPUT_G6_VAR.O_G6_GRIPPER_OPEN_4:=FALSE;
ELSE
	INPUT_G6_VAR.O_G6_GRIPPER_CLOSE_4:=FALSE;
	INPUT_G6_VAR.O_G6_GRIPPER_OPEN_4:=TRUE;
END_IF

//EXTENDER DOWN
IF INPUT_G6_VAR.IX_G6_GRIPPER_EXT_1 THEN
	INPUT_G6_VAR.O_G6_GRIPPER_EXT_DOWN_1:=TRUE;
	INPUT_G6_VAR.O_G6_GRIPPER_EXT_UP_1:=FALSE;
ELSE
	INPUT_G6_VAR.O_G6_GRIPPER_EXT_DOWN_1:=FALSE;
	INPUT_G6_VAR.O_G6_GRIPPER_EXT_UP_1:=TRUE;
END_IF

IF INPUT_G6_VAR.IX_G6_GRIPPER_EXT_2 THEN
	INPUT_G6_VAR.O_G6_GRIPPER_EXT_DOWN_2:=TRUE;
	INPUT_G6_VAR.O_G6_GRIPPER_EXT_UP_2:=FALSE;
ELSE
	INPUT_G6_VAR.O_G6_GRIPPER_EXT_DOWN_2:=FALSE;
	INPUT_G6_VAR.O_G6_GRIPPER_EXT_UP_2:=TRUE;
END_IF

IF INPUT_G6_VAR.IX_G6_GRIPPER_EXT_3 THEN
	INPUT_G6_VAR.O_G6_GRIPPER_EXT_DOWN_3:=TRUE;
	INPUT_G6_VAR.O_G6_GRIPPER_EXT_UP_3:=FALSE;
ELSE
	INPUT_G6_VAR.O_G6_GRIPPER_EXT_DOWN_3:=FALSE;
	INPUT_G6_VAR.O_G6_GRIPPER_EXT_UP_3:=TRUE;
END_IF

IF INPUT_G6_VAR.IX_G6_GRIPPER_EXT_4 THEN
	INPUT_G6_VAR.O_G6_GRIPPER_EXT_DOWN_4:=TRUE;
	INPUT_G6_VAR.O_G6_GRIPPER_EXT_UP_4:=FALSE;
ELSE
	INPUT_G6_VAR.O_G6_GRIPPER_EXT_DOWN_4:=FALSE;
	INPUT_G6_VAR.O_G6_GRIPPER_EXT_UP_4:=TRUE;
END_IF

TP_END_FUKUDA(IN:=INPUT_G6_VAR.I_G6_END_FUKUDA,PT:=T#0.1S);
CNT_END_FUKUDA(CU:=TP_END_FUKUDA.Q,RESET:=INPUT_G6_VAR.I_G6_ENABLE,PV:=10);
(*IF CNT_END_FUKUDA.CV MOD 2=1 THEN
	INPUT_G6_VAR.O_G6_SELECT_FUKUDA_A:=TRUE;
ELSE
	INPUT_G6_VAR.O_G6_SELECT_FUKUDA_A:=FALSE;
END_IF*)

//INPUT_G6_VAR.O_G6_SELECT_FUKUDA_A:=


INPUT_VAR.I_STOPPER_TRANSFER_ON_A:= INPUT_VAR.O_STOPPER_TRANSFER_A;
//IF INPUT_VAR.I_STOPPER_TRANSFER_ON_A OR INPUT_VAR.I_STOPPER_TRANSFER_ON_B THEN

INPUT_G6_VAR.O_G6_SETMOTORON:=TRUE;
TMR1(IN:=INPUT_G6_VAR.O_G6_SETMOTORON ,PT:=T#0.5S);
IF TMR1.Q THEN
	TP2(IN:=TMR1.Q,PT:=T#1S);
	INPUT_G6_VAR.O_G6_STOP:=TP2.Q;
	IF INPUT_G6_VAR.I_G6_READY THEN
		TP3(IN:=INPUT_G6_VAR.O_G6_SETMOTORON,PT:=T#0.1S);
		INPUT_G6_VAR.O_G6_HOME:=TP3.Q;
	END_IF
END_IF

IF INPUT_G6_VAR.O_G6_SETMOTORON AND INDEXING_1_VAR.I_INDEXING_1_ROTATION_DONE AND INDEXING_1_VAR.I_INDEXING_1_HOME THEN
	IF INPUT_G6_VAR.I_G6_READY OR INPUT_G6_VAR.I_G6_RUNNING THEN

// ERROR OVERRIDE
		IF 	INPUT_G6_VAR.I_G6_ERROR THEN
			TMR10(IN:=INPUT_G6_VAR.I_G6_ERROR,PT:=T#0.5S);
			IF NOT TMR10.Q THEN
				INPUT_G6_VAR.O_G6_RESET :=TRUE;	
				INPUT_G6_VAR.O_G6_START :=FALSE ;
				INPUT_G6_VAR.O_G6_CONTINUE :=FALSE;
				TMR10(IN:=FALSE);
			ELSE
				INPUT_G6_VAR.O_G6_RESET :=FALSE;		
			END_IF
		END_IF
	 
		//TMR8(IN:=INPUT_G6_VAR.O_G6_SELECT_FUKUDA_A,PT:=T#5S);
		//TMR9(IN:=INPUT_G6_VAR.O_G6_START,PT:=T#2S);
		
//START FOR 1ST TIME
		IF INPUT_G6_VAR.I_G6_READY AND NOT INPUT_G6_VAR.I_G6_ERROR AND NOT INPUT_G6_VAR.I_G6_RUNNING THEN
			TMR7(IN:=INPUT_G6_VAR.I_G6_READY,PT:=T#1S);
			START_ROBOT(IN:=TMR7.Q,PT:=T#2S);
			INPUT_G6_VAR.O_G6_START :=TMR7.Q ;
			INPUT_G6_VAR.O_G6_STOP:=FALSE;
		ELSE
			TMR7(IN:=FALSE);
		END_IF
		IF  NOT INPUT_G6_VAR.I_G6_READY THEN
			INPUT_G6_VAR.O_G6_START :=FALSE ;
		END_IF
		
//STOP 
		IF INPUT_G6_VAR.I_G6_END_FUKUDA AND NOT INPUT_G6_VAR.I_G6_READY AND NOT INPUT_G6_VAR.I_G6_RUNNING THEN
			TMR8(IN:=FALSE);
			TMR9(IN:=FALSE);
		//	INPUT_G6_VAR.O_G6_STOP:=TRUE;
		END_IF
		TMR2(IN:=INPUT_G6_VAR.O_G6_STOP,PT:=T#1S);
		IF TMR2.Q THEN
			INPUT_G6_VAR.I_G6_HANG:=FALSE;
			INPUT_G6_VAR.O_G6_STOP:=FALSE;
			TMR1(IN:=FALSE);
		END_IF
		
//CONTINUE	
		//INPUT_G6_VAR.GO_ROBOT:=(INPUT_G6_VAR.I_G6_READY_PLACING AND LOADER_RS4_VAR.I_LOADER_RS4_READY_TAKEUP AND INDEXING_2_VAR.O_ROTATION_DONE )OR(INPUT_G6_VAR.I_G6_READY_PLACING AND NOT LOADER_RS4_VAR.I_LOADER_RS4_ENABLE AND  INDEXING_1_VAR.I_INDEXING_1_ROTATION_DONE)    ;	
		IF (INPUT_G6_VAR.I_G6_READY_PLACING AND LOADER_RS4_VAR.I_LOADER_RS4_READY_TAKEUP AND  INDEXING_1_VAR.I_INDEXING_1_ROTATION_DONE AND INDEXING_2_VAR.O_ROTATION_DONE)  THEN
			INPUT_G6_VAR.GO_ROBOT:=TRUE;
		END_IF
		IF (INPUT_G6_VAR.I_G6_READY_PLACING AND NOT LOADER_RS4_VAR.I_LOADER_RS4_ENABLE AND  INDEXING_1_VAR.I_INDEXING_1_ROTATION_DONE AND INDEXING_2_VAR.O_ROTATION_DONE) THEN
			INPUT_G6_VAR.GO_ROBOT:=TRUE;
		END_IF
		IF INDEXING_1_VAR.I_INDEXING_1_ROTATION_DONE AND INPUT_G6_VAR.GO_ROBOT AND INPUT_VAR.STRAIGHTEN_DONE AND NOT INPUT_G6_VAR.I_G6_END_FUKUDA AND INPUT_G6_VAR.I_G6_RUNNING AND NOT LOADER_RS4_VAR.I_LOADER_RS4_END_CARRIER THEN
				TMR3(IN:=INPUT_G6_VAR.GO_ROBOT ,PT:=T#0.5S);
				TP1(IN:=INPUT_G6_VAR.GO_ROBOT,PT:=T#0.1S);
		ELSE
			TMR3(IN:=FALSE);
			TP1(IN:=FALSE);
		END_IF
		INPUT_G6_VAR.O_G6_CONTINUE :=TMR3.Q;

		CNT_CYCLE(CU:=INPUT_G6_VAR.I_G6_START_TAKEUP,RESET:=INPUT_G6_VAR.I_G6_DISABLE,PV:=4);
		IF CNT_CYCLE.CV >=4 THEN
			LOADER_RS4_VAR.I_LOADER_RS4_ENABLE:=TRUE;
		END_IF
		IF CNT_CYCLE.CV =3 THEN
			INPUT_G6_VAR.O_G6_CONTINUE :=TRUE;
		END_IF
		IF NOT LOADER_RS4_VAR.I_LOADER_RS4_ENABLE AND INPUT_G6_VAR.I_G6_START_TAKEUP  THEN
				INDEXING_1_VAR.O_ROTATION_START:=TRUE;
		END_IF
		IF INPUT_G6_VAR.I_G6_START_PLACING THEN
			INDEXING_1_VAR.O_ROTATION_START:=FALSE;
		END_IF
 
		IF INPUT_G6_VAR.I_G6_START_TAKEUP AND LOADER_RS4_VAR.I_LOADER_RS4_START_PLACING  THEN
			INPUT_G6_VAR.GO_ROBOT:=FALSE;
		END_IF
END_IF
END_IF
END_IF
//END_IF

END_PROGRAM

// ---- POUs/LOADER/INDEXING.TcPOU
PROGRAM INDEXING
VAR
	bStartInput : BOOL;
	bServoOn : BOOL;
	bProgram0_On : BOOL;
	bProgram1_On : BOOL :=TRUE;
	bProgram2_On : BOOL :=FALSE;
	bProgram3_On : BOOL:=FALSE;
	bProgram4_On : BOOL:=FALSE;	
	bHomePositionReturn : BOOL;
	bResetInput : BOOL;
	bEmergencyInput : BOOL := TRUE;
	
	IN_POSITION_INPUT: BOOL;
	IN_POSITIONING_COMPLETION: BOOL;
	IN_START_INPUT_WAIT: BOOL;
	IN_ALARM1: BOOL;
	IN_ALARM2: BOOL;
	IN_READY_STATE: BOOL;
	T1: TON;
	TMR1: TON;
	TMR2: TON;
	TMR3: TON;
	TMR4: TON;
	TMR5: TON;
	TMR6: TON;
	TMR7: TON;
	IN_SERVO_STATUS: BOOL;
	bFirstDigit: BOOL;
	CNT1: CTU;
	ResetCount: BOOL;
	IPC: TP;
	IN_POSITIONING_COMPLET: BOOL;
	CNT2: CTU;
	START_STRAIGTHEN: BOOL;

	START_STRAIGHTEN: R_TRIG;
	START_ROTATING: R_TRIG;
	START_ROTATION: TP;
	SS: R_TRIG;
	CNT_START: CTU;
	TMR_PROCESS: TOF;
END_VAR

INDEXING_1_VAR.DataByteOutput[0].0 := bProgram0_On;
INDEXING_1_VAR.DataByteOutput[0].1 := bProgram1_On;
INDEXING_1_VAR.DataByteOutput[0].2 := bProgram2_On;
INDEXING_1_VAR.DataByteOutput[0].3 := bProgram3_On;
INDEXING_1_VAR.DataByteOutput[0].4 := bProgram4_On;
INDEXING_1_VAR.DataByteOutput[0].6 := bResetInput;
INDEXING_1_VAR.DataByteOutput[0].7 := bHomePositionReturn;
INDEXING_1_VAR.DataByteOutput[1].0 := bStartInput;
INDEXING_1_VAR.DataByteOutput[1].1 := bServoOn;
INDEXING_1_VAR.DataByteOutput[1].2 := bFirstDigit;
INDEXING_1_VAR.DataByteOutput[1].4 := bEmergencyInput;

IN_POSITION_INPUT := 			INDEXING_1_VAR.DataByteInput [1].0;
IN_POSITIONING_COMPLETION := 	INDEXING_1_VAR.DataByteInput [1].1;
IN_START_INPUT_WAIT := 			INDEXING_1_VAR.DataByteInput [1].2;
IN_ALARM1 := 					INDEXING_1_VAR.DataByteInput [1].3;
IN_ALARM2 := 					INDEXING_1_VAR.DataByteInput [1].4;
IN_READY_STATE :=				INDEXING_1_VAR.DataByteInput [1].7;
IN_SERVO_STATUS :=				INDEXING_1_VAR.DataByteInput [1].6; 

//ALARM RESET
IF IN_ALARM1 OR IN_ALARM2 THEN
	bResetInput := TRUE;
	TMR4(IN:=bResetInput,PT:=T#0.5S);
	IF TMR4.Q THEN
		bResetInput := FALSE;
	END_IF
ELSE
	TMR4(IN:=FALSE);
END_IF

IF NOT INDEXING_1_VAR.I_INDEXING_1_HOME THEN
	INDEXING_1_VAR.O_INDEXING_1_HOME:=TRUE;
 	ResetCount:=TRUE;
	INDEXING_1_VAR.O_ROTATION_START:=FALSE;
 	IF IN_POSITIONING_COMPLET THEN
		INDEXING_1_VAR.I_INDEXING_1_HOME:=TRUE;
	END_IF
END_IF

IF INDEXING_1_VAR.O_INDEXING_1_HOME THEN
	bHomePositionReturn:=TRUE;
	IF IN_POSITIONING_COMPLET THEN
		INDEXING_1_VAR.O_INDEXING_1_HOME:=FALSE;
		bHomePositionReturn:=FALSE;
	END_IF
END_IF

START_ROTATING(CLK:=INDEXING_1_VAR.O_ROTATION_START);
IF INDEXING_1_VAR.O_ROTATION_START AND IN_START_INPUT_WAIT AND INDEXING_1_VAR.I_INDEXING_1_HOME AND INPUT_VAR.STRAIGHTEN_DONE  THEN
	INDEXING_1_VAR.READY_STRAIGTHEN:=TRUE;
	ELSE
	INDEXING_1_VAR.READY_STRAIGTHEN:=FALSE;	
END_IF

START_ROTATION(IN:=INDEXING_1_VAR.READY_STRAIGTHEN,PT:=T#0.1S);
IF 	START_ROTATION.Q AND NOT TMR_PROCESS.Q AND INDEXING_1_VAR.I_PRESS_STOPPER_UP AND INPUT_VAR.STRAIGHTEN_DONE AND NOT INPUT_G6_VAR.I_G6_START_PLACING AND NOT LOADER_RS4_VAR.I_LOADER_RS4_START_TAKEUP THEN
	bprogram0_on:=TRUE;
	IF bprogram0_on THEN
		INDEXING_1_VAR.O_ROTATION_START:=FALSE;
	END_IF
	
	INDEXING_1_VAR.I_INDEXING_1_ROTATION_DONE:=FALSE;
	IN_POSITIONING_COMPLET :=FALSE;
END_IF
IF bprogram0_on THEN
	TMR_PROCESS(IN:=TRUE,PT:=T#3S);
	INDEXING_1_VAR.O_ROTATION_START:=FALSE;
ELSE
	TMR_PROCESS(IN:=FALSE);
END_IF
//select Program No.
IF bprogram0_on AND INDEXING_1_VAR.I_PRESS_STOPPER_UP AND NOT INPUT_G6_VAR.I_G6_START_PLACING AND NOT LOADER_RS4_VAR.I_LOADER_RS4_START_TAKEUP  THEN
	INDEXING_1_VAR.O_ROTATION_START:=FALSE;
	TMR1(IN:=bprogram0_on,PT:=T#15MS);
	bStartInput:=tmr1.Q ;
	IF tmr1.Q THEN
		TMR2(in:=TRUE,pt:=T#25MS);
	END_IF
	
	IF tmr2.Q THEN
		tmr1(in:=FALSE);
		bStartInput:=FALSE;
	END_IF
	tmr3(in:=tmr2.
Q,pt:=T#5MS);
	IF tmr3.Q THEN
		bprogram0_on:= FALSE;
		tmr2(in:=FALSE);
		tmr3(in:=FALSE);
	END_IF
END_IF

IPC(IN:=IN_POSITIONING_COMPLETION,PT:=T#0.4S);
IF IPC.Q THEN
	IN_POSITIONING_COMPLET :=TRUE;
END_IF
IF 	IN_POSITIONING_COMPLET THEN
	INDEXING_1_VAR.I_INDEXING_1_ROTATION_DONE:=TRUE;
END_IF
IF INDEXING_1_VAR.I_PRESS_STOPPER_UP AND INDEXING_1_VAR.I_INDEXING_1_ROTATION_DONE THEN
	SS(CLK:=INDEXING_1_VAR.I_INDEXING_1_ROTATION_DONE );
	CNT_START(CU:=SS.Q,RESET:= CNT_START.Q,PV:=2);
	IF CNT_START.CV=1 THEN
	INPUT_VAR.STRAIGHTEN_START:=SS.Q;
	END_IF
	IN_POSITIONING_COMPLET :=FALSE;
	ELSE
SS(CLK:=FALSE);
END_IF
(*
 IF CNT2.CV >=2 THEN
	 bprogram0_on:=FALSE;
	 bStartInput:=FALSE;
 END_IF

CNT1(CU:=IN_POSITIONING_COMPLET,RESET:=ResetCount,PV:=4);
CNT2(CU:=bprogram0_on,RESET:=ResetCount,PV:=2);
TMR5(IN:=CNT1.Q,PT:=T#0.5S);

IF TMR5.Q AND INDEXING_1_VAR.I_PRESS_STOPPER_UP THEN
	INDEXING_1_VAR.O_ROTATION_START:=TRUE;
	ResetCount:=TRUE;
	TMR5(IN:=FALSE);
ELSE
	ResetCount:=FALSE;
END_IF
*)

END_PROGRAM

// ---- POUs/LOADER/INDEXING_2.TcPOU
PROGRAM INDEXING_2
VAR
	bStartInput : BOOL;
	bServoOn : BOOL;
	bProgram0_On : BOOL;
	bProgram1_On : BOOL :=TRUE;
	bProgram2_On : BOOL :=FALSE;
	bProgram3_On : BOOL:=FALSE;
	bProgram4_On : BOOL:=FALSE;	
	bHomePositionReturn : BOOL;
	bResetInput : BOOL;
	bEmergencyInput : BOOL := TRUE;
	
	IN_POSITION_INPUT: BOOL;
	IN_POSITIONING_COMPLETION: BOOL;
	IN_START_INPUT_WAIT: BOOL;
	IN_ALARM1: BOOL;
	IN_ALARM2: BOOL;
	IN_READY_STATE: BOOL;
	T1: TON;
	TMR1: TON;
	TMR2: TON;
	TMR3: TON;
	TMR4: TON;
	TMR5: TON;
	TMR6: TON;
	TMR7: TON;
	IN_SERVO_STATUS: BOOL;
	CNT1: CTU;
	ENABLE_TIMER: INT;
	ResetCount: BOOL;
	CNT_INDEX: CTU;
	
	RESET_CNT_INDEX: BOOL;
END_VAR

INDEXING_2_VAR.DataByteOutput2[0].0 := bProgram0_On;
INDEXING_2_VAR.DataByteOutput2[0].1 := bProgram1_On;
INDEXING_2_VAR.DataByteOutput2[0].2 := bProgram2_On;
INDEXING_2_VAR.DataByteOutput2[0].3 := bProgram3_On;
INDEXING_2_VAR.DataByteOutput2[0].4 := bProgram4_On;
INDEXING_2_VAR.DataByteOutput2[0].6 := bResetInput;
INDEXING_2_VAR.DataByteOutput2[0].7 := bHomePositionReturn;
INDEXING_2_VAR.DataByteOutput2[1].0 := bStartInput;
INDEXING_2_VAR.DataByteOutput2[1].1 := bServoOn;
INDEXING_2_VAR.DataByteOutput2[1].4 := bEmergencyInput;

IN_POSITION_INPUT := INDEXING_2_VAR.DataByteInput2 [1].0;
IN_POSITIONING_COMPLETION := INDEXING_2_VAR.DataByteInput2 [1].1;
IN_START_INPUT_WAIT := INDEXING_2_VAR.DataByteInput2 [1].2;
IN_ALARM1 := INDEXING_2_VAR.DataByteInput2 [1].3;
IN_ALARM2 := INDEXING_2_VAR.DataByteInput2 [1].4;
IN_READY_STATE :=INDEXING_2_VAR.DataByteInput2 [1].7;
IN_SERVO_STATUS :=INDEXING_2_VAR.DataByteInput2 [1].6; 

//ALARM RESET
IF IN_ALARM1 OR IN_ALARM2 THEN
	bResetInput := TRUE;
	TMR4(IN:=bResetInput,PT:=T#0.5S);
	IF TMR4.Q THEN
		bResetInput := FALSE;
	END_IF
ELSE
	TMR4(IN:=FALSE);
END_IF

IF NOT INDEXING_2_VAR.I_INDEXING_2_HOME THEN
 	INDEXING_2_VAR.O_INDEXING_HOME:=TRUE;
 	IF IN_POSITIONING_COMPLETION THEN
		INDEXING_2_VAR.I_INDEXING_2_HOME:=TRUE;
	END_IF
END_IF
 
IF INDEXING_2_VAR.O_INDEXING_HOME THEN
	bHomePositionReturn:=TRUE;
	ResetCount:=TRUE;
	INDEXING_2_VAR.O_ROTATION_START:=FALSE;
	RESET_CNT_INDEX:=TRUE;
	IF IN_POSITIONING_COMPLETION THEN
		INDEXING_2_VAR.O_INDEXING_HOME:=FALSE;
		bHomePositionReturn:=FALSE;
			
	END_IF
ELSE
	RESET_CNT_INDEX:=FALSE;
END_IF

IF 	INDEXING_2_VAR.O_ROTATION_START AND IN_START_INPUT_WAIT AND NOT INDEXING_2_VAR.O_INDEXING_HOME THEN
	bprogram0_on:=TRUE;
	INDEXING_2_VAR.O_ROTATION_DONE:=FALSE;
END_IF

//select Program No.
IF bprogram0_on THEN
	INDEXING_2_VAR.O_ROTATION_START:=FALSE;
	TMR1(IN:=bprogram0_on,PT:=T#15MS);
	bStartInput:=tmr1.Q ;
	IF tmr1.Q THEN
		TMR2(in:=TRUE,pt:=T#25MS);
	END_IF
	
	IF tmr2.Q THEN
		tmr1(in:=FALSE);
		bStartInput:=FALSE;
	END_IF
	tmr3(in:=tmr2.Q,pt:=T#5MS);
	IF tmr3.Q THEN
		bprogram0_on:= FALSE;
		tmr2(in:=FALSE);
		tmr3(in:=FALSE);
	END_IF
END_IF
IF  INDEXING_2_VAR.I_INDEXING_2_HOME THEN
	CNT_INDEX(CU:=bprogram0_on,RESET:=CNT_INDEX.Q,PV:=4);
	ELSE
	CNT_INDEX(CU:=FALSE);
	INDEXING_2_VAR.CARRIER_INDEX :=100;
END_IF

CASE CNT_INDEX.CV OF
	0:
	INDEXING_2_VAR.CARRIER_INDEX :=0;
	RESET_CNT_INDEX:=FALSE;
	1:
	INDEXING_2_VAR.CARRIER_INDEX :=1;
	2:
	INDEXING_2_VAR.CARRIER_INDEX :=2;
	3:
	INDEXING_2_VAR.CARRIER_INDEX :=3;
ELSE
	INDEXING_2_VAR.CARRIER_INDEX :=0;
END_CASE

IF RESET_CNT_INDEX THEN
	CNT_INDEX(CU:=FALSE);
END_IF
IF 	IN_POSITIONING_COMPLETION THEN
	INDEXING_2_VAR.O_ROTATION_DONE:=TRUE;
	INDEXING_2_VAR.O_ROTATION_START:=FALSE;
	LOADER_RS4_VAR.I_LOADER_RS4_END_CARRIER:=FALSE;
END_IF
(*
CNT1(CU:=IN_POSITIONING_COMPLETION,RESET:=ResetCount,PV:=4);
TMR5(IN:=CNT1.Q,PT:=T#0.5S);

IF TMR5.Q THEN
	INDEXING_2_VAR.O_ROTATION_START:=TRUE;
	ResetCount:=TRUE;
	TMR5(IN:=FALSE);
ELSE
		ResetCount:=FALSE;
END_IF
 *)

END_PROGRAM

// ---- POUs/INPUT_PROG.TcPOU
PROGRAM INPUT_PROG
VAR
	T1: TON;
	
	T2: TON;
	Q: BOOL;
	OUT1: BOOL;
	AR: R_TRIG;
	LOTBOX_STAT: BOOL;
	RTRIG_1: F_TRIG;
	RTRIG_2: F_TRIG;
	RTRIG_3: F_TRIG;
	RTRIG_4: F_TRIG;
	QUEUE_INDEX_1: INT;
	QUEUE_INDEX_2: INT;
	QUEUE_INDEX_3: INT;
	QUEUE_INDEX_4: INT;
	IC_CASE: INT;
	TMR1: TON;
	TMR2: TON;
	I_STOPPER_TRANSFER_A: INT;
	TMR3: TON;
	TMR4: TON;
	TMR5: TON;
	TMR6: TON;
	TMR7: TON;
	TMR8: TON;
	TMR9: TON;
	TMR10: TON;
	TMR11: TON;
	TMR12: TON;
	TMR14: TON;
	COUNTER_1: CTU;
	RESET_COUNTER: BOOL;
	COUNTER_2: CTU;
END_VAR

VAR PERSISTENT
	AR_TRIG: R_TRIG;
END_VAR


//INDICATOR LOTBOX
INPUT_VAR.O_LOT_BOX_INDICATOR_1:= NOT INPUT_VAR.I_LOTBOX_DETECT_1;
INPUT_VAR.O_LOT_BOX_INDICATOR_2:= NOT INPUT_VAR.I_LOTBOX_DETECT_2;
INPUT_VAR.O_LOT_BOX_INDICATOR_3:= NOT INPUT_VAR.I_LOTBOX_DETECT_3;
INPUT_VAR.O_LOT_BOX_INDICATOR_4:= NOT INPUT_VAR.I_LOTBOX_DETECT_4;

IF NOT INPUT_VAR.I_LOTBOX_DETECT_1 OR NOT INPUT_VAR.I_LOTBOX_DETECT_2 OR NOT INPUT_VAR.I_LOTBOX_DETECT_3 OR NOT INPUT_VAR.I_LOTBOX_DETECT_4 THEN
	INPUT_VAR.O_TOWER_LAMP_YELLOW :=TRUE;
END_IF 


IF FLAG_VAR.ALLOW_EXECUTE_LOAD_FUKUDA THEN 
	IF INPUT_VAR.I_CASE=100 OR INPUT_VAR.I_CASE=12 THEN
		INPUT_VAR.I_CASE:=0;
		IC_CASE:=0;	
		END_IF			
	LOAD_FUKUDA();
END_IF
IF FLAG_VAR.ALLOW_EXECUTE_RETURN_FUKUDA THEN 
	IF INPUT_VAR.I_CASE=100 THEN
		INPUT_VAR.I_CASE:=0;
		IC_CASE:=0;
	END_IF	
	RETURN_FUKUDA();	
END_IF

(*
TMR4(IN:=INPUT_VAR.I_FUKUDA_TRANSFER_AT_FRONT_B,PT:= T#2S);
TMR5(IN:=INPUT_VAR.I_STOPPER_TRANSFER_ON_B,PT:=T#2S);
TMR6(IN:=INPUT_G6_VAR.O_G6_SELECT_FUKUDA_B,PT:=T#10S);

INPUT_VAR.O_STOPPER_TRANSFER_B:=TMR4.Q;
INPUT_G6_VAR.O_G6_SELECT_FUKUDA_B:=TMR5.Q;
*)

//END_IF
//LOTBOX_STAT := INPUT_VAR.I_LOTBOX_DETECT_1 + INPUT_VAR.I_LOTBOX_DETECT_2 + INPUT_VAR.I_LOTBOX_DETECT_3 + INPUT_VAR.I_LOTBOX_DETECT_4 


//INPUT_G6_VAR.I_G6_HOME:=POWER_CONTROL.O_PWR_CTRL_ROBOT_G6;
//INDEXING1_VAR.I_INDEXING_HOME := POWER_CONTROL.O_PWR_CTRL_INDEXING_1;

RTRIG_1(CLK :=INPUT_VAR.I_LOTBOX_DETECT_1);
RTRIG_2(CLK :=INPUT_VAR.I_LOTBOX_DETECT_2);
RTRIG_3(CLK :=INPUT_VAR.I_LOTBOX_DETECT_3);
RTRIG_4(CLK :=INPUT_VAR.I_LOTBOX_DETECT_4);
(*
IF RTRIG_1.Q THEN
	IF QUEUE_INDEX_1 =0  THEN
		QUEUE_INDEX_1 :=1;
	ELSIF QUEUE_INDEX_2 =0 THEN
		QUEUE_INDEX_2 :=1;
	ELSIF QUEUE_INDEX_3 =0 THEN
		QUEUE_INDEX_3 :=1;
	ELSIF QUEUE_INDEX_4 =0 THEN
		QUEUE_INDEX_4 :=1;
	END_IF	
	INPUT_VAR.O_LOTBOX_CLAMP_ON_1:=TRUE;
	INPUT_VAR.O_LOTBOX_CLAMP_OFF_1:=FALSE;
ELSIF RTRIG_2.Q THEN
	IF QUEUE_INDEX_1 =0  THEN
		QUEUE_INDEX_1 :=2;
	ELSIF QUEUE_INDEX_2 =0 THEN
		QUEUE_INDEX_2 :=2;
	ELSIF QUEUE_INDEX_3 =0 THEN
		QUEUE_INDEX_3 :=2;
	ELSIF QUEUE_INDEX_4 =0 THEN
		QUEUE_INDEX_4 :=2;
	END_IF
	INPUT_VAR.O_LOTBOX_CLAMP_ON_2:=TRUE;
	INPUT_VAR.O_LOTBOX_CLAMP_OFF_2:=FALSE;
ELSIF RTRIG_3.Q THEN
	IF QUEUE_INDEX_1 =0  THEN
		QUEUE_INDEX_1 :=3;
	ELSIF QUEUE_INDEX_2 =0 THEN
		QUEUE_INDEX_2 :=3;
	ELSIF QUEUE_INDEX_3 =0 THEN
		QUEUE_INDEX_3 :=3;
	ELSIF QUEUE_INDEX_4 =0 THEN
		QUEUE_INDEX_4 :=3;
	END_IF	
	INPUT_VAR.O_LOTBOX_CLAMP_ON_3:=TRUE;
	INPUT_VAR.O_LOTBOX_CLAMP_OFF_3:=FALSE;
ELSIF RTRIG_4.Q THEN
	IF QUEUE_INDEX_1 =0  THEN
		QUEUE_INDEX_1 :=4;
	ELSIF QUEUE_INDEX_2 =0 THEN
		QUEUE_INDEX_2 :=4;
	ELSIF QUEUE_INDEX_3 =0 THEN
		QUEUE_INDEX_3 :=4;
	ELSIF QUEUE_INDEX_4 =0 THEN
		QUEUE_INDEX_4 :=4;
	END_IF	
	INPUT_VAR.O_LOTBOX_CLAMP_ON_4:=TRUE;
	INPUT_VAR.O_LOTBOX_CLAMP_OFF_4:=FALSE;	
END_IF

IF NOT INPUT_VAR.I_LOTBOX_DETECT_1 THEN
	QUEUE_INDEX_1 :=0;
END_IF
IF NOT INPUT_VAR.I_LOTBOX_DETECT_2 THEN
	QUEUE_INDEX_2 :=0;
END_IF
IF NOT INPUT_VAR.I_LOTBOX_DETECT_3 THEN
	QUEUE_INDEX_3 :=0;
END_IF
IF NOT INPUT_VAR.I_LOTBOX_DETECT_4 THEN
	QUEUE_INDEX_4 :=0;
END_IF

IF INPUT_VAR.I_LOTEND THEN
	INPUT_VAR.O_LOTBOX_CLAMP_ON_1:=FALSE;
	INPUT_VAR.O_LOTBOX_CLAMP_ON_2:=FALSE;
	INPUT_VAR.O_LOTBOX_CLAMP_ON_3:=FALSE;
	INPUT_VAR.O_LOTBOX_CLAMP_ON_4:=FALSE;
	INPUT_VAR.O_LOTBOX_CLAMP_OFF_1:=TRUE;
	INPUT_VAR.O_LOTBOX_CLAMP_OFF_2:=TRUE;
	INPUT_VAR.O_LOTBOX_CLAMP_OFF_3:=TRUE;
	INPUT_VAR.O_LOTBOX_CLAMP_OFF_4:=TRUE;
			
END_IF
*)	
 
(*
INPUT_VAR.O_STOPPER_TRANSFER_A:=TMR11.Q ;
INPUT_VAR.O_STOPPER_TRANSFER_B:=TMR12.Q ;

TMR14(IN:=INPUT_G6_VAR.I_G6_END_FUKUDA,PT:=T#10S);
IF NOT TMR14.Q AND INPUT_G6_VAR.I_G6_END_FUKUDA THEN
	TMR11(IN:=FALSE);
	TMR12(IN:=FALSE);
ELSE
	TMR11(IN:=INPUT_VAR.I_FUKUDA_TRANSFER_AT_FRONT_A,PT:=T#2S);	
	TMR12(IN:=INPUT_VAR.I_FUKUDA_TRANSFER_AT_FRONT_B,PT:=T#2S);

END_IF
 

 IF INPUT_G6_VAR.I_G6_END_FUKUDA AND NOT INPUT_VAR.ACTIVE_PROGRAM_CHANGE THEN
	INPUT_VAR.ACTIVE_PROGRAM:=INPUT_VAR.ACTIVE_PROGRAM+1;
	IF INPUT_VAR.ACTIVE_PROGRAM=3 THEN
		INPUT_VAR.ACTIVE_PROGRAM:=1;
	END_IF
	INPUT_VAR.ACTIVE_PROGRAM_CHANGE:=TRUE;
 END_IF

 COUNTER_1(CU:=INPUT_G6_VAR.I_G6_END_CYCLE,RESET:=INPUT_G6_VAR.O_G6_START,PV:=14);
IF COUNTER_1.CV =1 THEN
	INPUT_VAR.ACTIVE_PROGRAM_CHANGE:=FALSE;
END_IF
 
*)

END_PROGRAM

// ---- POUs/FUKUDA/LOAD_FUKUDA.TcPOU
PROGRAM LOAD_FUKUDA
VAR_INPUT

END_VAR

VAR
	TMR_DELAY: TON;
	TMR1:TON;
	TMR_STOPPER_A: TON;
	TMR_STOPPER_B: TON;
END_VAR

CASE INPUT_VAR.I_CASE OF
0: //standby near lotbox
	IF INPUT_VAR.ACTIVE_ID=6 THEN
		INPUT_VAR.ACTIVE_ID:=1;
	END_IF
	CASE INPUT_VAR.I_CURRENT_TRANSACTION.TRANSPORT_INDEX OF
		2 : FUKUDA_MOVE(STEP_DATA_1:=INPUT_VAR.I_CURRENT_TRANSACTION.STATION_NUMBER_LOAD,
				STEP_DATA_2:=3,
				STEP_DATA_3:=INPUT_VAR.I_CURRENT_TRANSACTION.JIG_INDEX_LOAD,
				STEP_DATA_4:=0,
				STEP_DATA_5:=1);
				INPUT_VAR.O_STOPPER_TRANSFER_B:=FALSE;
		1 : FUKUDA_MOVE(STEP_DATA_1:=INPUT_VAR.I_CURRENT_TRANSACTION.STATION_NUMBER_LOAD,
				STEP_DATA_2:=3,
				STEP_DATA_3:=INPUT_VAR.I_CURRENT_TRANSACTION.JIG_INDEX_LOAD,
				STEP_DATA_4:=1,
				STEP_DATA_5:=0);
				INPUT_VAR.O_STOPPER_TRANSFER_A:=FALSE;
	END_CASE			
	input_var.O_VACUUM_On:=FALSE;
	input_var.O_VACUUM_OFF:=FALSE;	
	
			
1: //standby near lotbox
	
	IF INPUT_VAR.ACTIVE_ID=6 THEN
		INPUT_VAR.ACTIVE_ID:=1;
	END_IF
		FUKUDA_MOVE(STEP_DATA_1:=INPUT_VAR.I_CURRENT_TRANSACTION.STATION_NUMBER_LOAD,
				STEP_DATA_2:=4,
				STEP_DATA_3:=INPUT_VAR.I_CURRENT_TRANSACTION.JIG_INDEX_LOAD,
				STEP_DATA_4:=0,
				STEP_DATA_5:=0);

		CASE INPUT_VAR.I_CURRENT_TRANSACTION.TRANSPORT_INDEX OF
		1:
			INPUT_VAR.I_LOADING_DONE_A:=FALSE;
		
		2:
			INPUT_VAR.I_LOADING_DONE_B:=FALSE;
	END_CASE
	
				
2://vacuum position 
	IF INPUT_VAR.ACTIVE_ID=6 THEN
		INPUT_VAR.ACTIVE_ID:=1;
	END_IF
	INPUT_VAR.I_CASE:=INPUT_VAR.I_CASE+1;
	(*FUKUDA_MOVE(STEP_DATA_1:=INPUT_VAR.I_CURRENT_TRANSACTION.STATION_NUMBER_LOAD,
				STEP_DATA_2:=4,
				STEP_DATA_3:=INPUT_VAR.I_CURRENT_TRANSACTION.JIG_INDEX_LOAD,
				STEP_DATA_4:=0,
				STEP_DATA_5:=0);
	IF INPUT_VAR.ACTIVE_ID=3 THEN
		input_var.O_VACUUM_ON:=TRUE;
		input_var.O_VACUUM_OFF:=FALSE;	
	END_IF
	*)

3://vacuum position 
	IF INPUT_VAR.ACTIVE_ID=6 THEN
		INPUT_VAR.ACTIVE_ID:=1; 
	END_IF
	//INPUT_VAR.I_CASE:=INPUT_VAR.I_CASE+1;
	//IF INPUT_VAR.O_VACUUM_ON THEN
		FUKUDA_MOVE(STEP_DATA_1:=INPUT_VAR.I_CURRENT_TRANSACTION.STATION_NUMBER_LOAD,
				STEP_DATA_2:=4,
				STEP_DATA_3:=INPUT_VAR.I_CURRENT_TRANSACTION.JIG_INDEX_LOAD,
				STEP_DATA_4:=0,
				STEP_DATA_5:=0);
	//ELSE
		
	//END_IF
4://vacuum position 
	IF INPUT_VAR.ACTIVE_ID=6 THEN
		INPUT_VAR.ACTIVE_ID:=1;
	END_IF
	input_var.O_VACUUM_ON:=TRUE;
	input_var.O_VACUUM_OFF:=FALSE;
	 
	//CHECK JIG FUKUDA PRESENCE			
//	IF  input_var.O_VACUUM_ON THEN
//		TMR1(IN:=TRUE,PT:=T#2S);
//		IF TMR1.Q THEN
			//IF NOT INPUT_VAR.I_VACUUM_ON AND input_var.O_VACUUM_ON THEN
			//	INPUT_VAR.JIG_FUKUDA_PRESENCE :=TRUE;
				
				(*FUKUDA_MOVE(STEP_DATA_1:=7,
				STEP_DATA_2:=4,
				STEP_DATA_3:=INPUT_VAR.I_CURRENT_TRANSACTION.JIG_INDEX_LOAD,
				STEP_DATA_4:=0,
				STEP_DATA_5:=0);*)
			//ELSE
				INPUT_VAR.JIG_FUKUDA_PRESENCE :=FALSE;	
				FUKUDA_MOVE(STEP_DATA_1:=INPUT_VAR.I_CURRENT_TRANSACTION.STATION_NUMBER_LOAD,
				STEP_DATA_2:=2,
				STEP_DATA_3:=INPUT_VAR.I_CURRENT_TRANSACTION.JIG_INDEX_LOAD,
				STEP_DATA_4:=0,
				STEP_DATA_5:=0);
				
(*				FUKUDA_MOVE(STEP_DATA_1:=INPUT_VAR.I_CURRENT_TRANSACTION.STATION_NUMBER_LOAD,
				STEP_DATA_2:=1,
				STEP_DATA_3:=INPUT_VAR.I_CURRENT_TRANSACTION.JIG_INDEX_LOAD,
				STEP_DATA_4:=0,
				STEP_DATA_5:=0);
				
				TMR_DELAY(IN:=TRUE,PT:=T#2S);
				IF TMR_DELAY.Q THEN
					FLAG_VAR.ALLOW_EXECUTE_LOAD_FUKUDA:=FALSE;
					INPUT_VAR.I_CURRENT_TRANSACTION.JIG_INDEX_LOAD:=INPUT_VAR.I_CURRENT_TRANSACTION.JIG_INDEX_LOAD+0;
					INPUT_VAR.I_CASE:=0;
					TMR1(IN:=FALSE);
					input_var.O_VACUUM_ON:=FALSE;
					input_var.O_VACUUM_OFF:=FALSE;
				END_IF
			//END_IF
		END_IF 
	END_IF 
*)
				

5://vacuum position 
	IF INPUT_VAR.ACTIVE_ID=6 THEN
		INPUT_VAR.ACTIVE_ID:=1;
	END_IF
	
	FUKUDA_MOVE(STEP_DATA_1:=8,
				STEP_DATA_2:=2,
				STEP_DATA_3:=INPUT_VAR.I_CURRENT_TRANSACTION.JIG_INDEX_LOAD,
				STEP_DATA_4:=0,
				STEP_DATA_5:=0);
	
6://gripping position
	IF INPUT_VAR.ACTIVE_ID=6 THEN
		INPUT_VAR.ACTIVE_ID:=1;
	END_IF

	FUKUDA_MOVE(STEP_DATA_1:=INPUT_VAR.I_CURRENT_TRANSACTION.TRANSPORT_INDEX+4,
				STEP_DATA_2:=2,
				STEP_DATA_3:=12,
				STEP_DATA_4:=0,
				STEP_DATA_5:=0);


7://placing onto fukuda transport
	IF INPUT_VAR.ACTIVE_ID=6 THEN
		INPUT_VAR.ACTIVE_ID:=1;
	END_IF
	FUKUDA_MOVE(STEP_DATA_1:=INPUT_VAR.I_CURRENT_TRANSACTION.TRANSPORT_INDEX+4,
				STEP_DATA_2:=2,
				STEP_DATA_3:=11,
				STEP_DATA_4:=0,
				STEP_DATA_5:=0);

8://placing onto fukuda transport
	IF INPUT_VAR.ACTIVE_ID=6 THEN
		INPUT_VAR.ACTIVE_ID:=1;
	END_IF
	
	FUKUDA_MOVE(STEP_DATA_1:=INPUT_VAR.I_CURRENT_TRANSACTION.TRANSPORT_INDEX+4,
				STEP_DATA_2:=2,
				STEP_DATA_3:=11,
				STEP_DATA_4:=0,
				STEP_DATA_5:=0);
	(*IF INPUT_VAR.ACTIVE_ID=3 THEN
		input_var.O_VACUUM_On:=FALSE;
		input_var.O_VACUUM_OFF:=TRUE;	
	END_IF
	*)
	
9://homing
	IF INPUT_VAR.ACTIVE_ID=6 THEN
		INPUT_VAR.ACTIVE_ID:=1;
	END_IF
	IF INPUT_VAR.I_VACUUM_ON THEN
		FUKUDA_MOVE(STEP_DATA_1:=INPUT_VAR.I_CURRENT_TRANSACTION.TRANSPORT_INDEX+4,
				STEP_DATA_2:=1,
				STEP_DATA_3:=13,//11
				STEP_DATA_4:=0,
				STEP_DATA_5:=0);
	ELSE
		input_var.O_VACUUM_On:=FALSE;
		input_var.O_VACUUM_OFF:=TRUE;
	END_IF	
				
10://pusH fukuda transport
	IF INPUT_VAR.ACTIVE_ID=6 THEN
		INPUT_VAR.ACTIVE_ID:=1;
	END_IF
	input_var.O_VACUUM_OFF:=FALSE;
	CASE INPUT_VAR.I_CURRENT_TRANSACTION.TRANSPORT_INDEX OF
		2 :
			IF NOT INPUT_VAR.I_FUKUDA_TRANSFER_AT_FRONT_B THEN
				FUKUDA_MOVE(STEP_DATA_1:=0,
				STEP_DATA_2:=0,
				STEP_DATA_3:=0,
				STEP_DATA_4:=0,
				STEP_DATA_5:=2);
			END_IF
				 
		1 : 
			IF NOT INPUT_VAR.I_FUKUDA_TRANSFER_AT_FRONT_A THEN
				FUKUDA_MOVE(STEP_DATA_1:=0,
				STEP_DATA_2:=0,
				STEP_DATA_3:=0,
				STEP_DATA_4:=2,
				STEP_DATA_5:=0);
			END_IF
	END_CASE			 
11:
				CASE INPUT_VAR.I_CURRENT_TRANSACTION.TRANSPORT_INDEX OF
		1:	
			IF INPUT_VAR.I_FUKUDA_TRANSFER_AT_FRONT_A THEN
				TMR_STOPPER_A(IN:=TRUE,PT:=T#0.8S);
				IF TMR_STOPPER_A.Q THEN 
					INPUT_VAR.O_STOPPER_TRANSFER_A:=TRUE;
					INPUT_VAR.I_LOADING_DONE_A:=TRUE;
					TMR1(IN:=FALSE);
					TMR_DELAY(IN:=FALSE);
					input_var.O_VACUUM_On:=FALSE;
					input_var.O_VACUUM_OFF:=TRUE;
					FLAG_VAR.ALLOW_EXECUTE_LOAD_FUKUDA:=FALSE;
					INPUT_G6_VAR.I_G6_ENABLE:=TRUE;
					INPUT_VAR.I_CASE:=100;
				END_IF
				
			ELSE
				TMR_STOPPER_A(IN:=FALSE);
				FUKUDA_MOVE(STEP_DATA_1:=0,
				STEP_DATA_2:=0,
				STEP_DATA_3:=0,
				STEP_DATA_4:=2,
				STEP_DATA_5:=0);
			END_IF 
			
			2:
			IF INPUT_VAR.I_FUKUDA_TRANSFER_AT_FRONT_B THEN
				
				TMR_STOPPER_B(IN:=TRUE,PT:=T#0.8S);
				IF TMR_STOPPER_B.Q THEN
					INPUT_VAR.O_STOPPER_TRANSFER_B:=TRUE;	
					INPUT_VAR.I_LOADING_DONE_B:=TRUE;
					TMR1(IN:=FALSE);
					TMR_DELAY(IN:=FALSE);
					input_var.O_VACUUM_On:=FALSE;
					input_var.O_VACUUM_OFF:=TRUE;
					FLAG_VAR.ALLOW_EXECUTE_LOAD_FUKUDA:=FALSE;
					INPUT_G6_VAR.I_G6_ENABLE:=TRUE;
					INPUT_VAR.I_CASE:=100;
				END_IF
			ELSE
				TMR_STOPPER_B(IN:=FALSE);
				FUKUDA_MOVE(STEP_DATA_1:=0,
				STEP_DATA_2:=0,
				STEP_DATA_3:=0,
				STEP_DATA_4:=0,
				STEP_DATA_5:=2);
			END_IF
			
	END_CASE
100:
	
	FLAG_VAR.ALLOW_EXECUTE_LOAD_FUKUDA:=FALSE;								
								
END_CASE

END_PROGRAM

// ---- POUs/FUKUDA/FUKUDA_MOVE.TcPOU
PROGRAM FUKUDA_MOVE
//FUNCTION FUKUDA_MOVE : BOOL
VAR_INPUT
	STEP_DATA_1: BYTE;
	STEP_DATA_2: BYTE;
	STEP_DATA_3: BYTE;
	STEP_DATA_4: BYTE;
	STEP_DATA_5: BYTE;
	FUKUDA_HOME: INT;
END_VAR

VAR
	
	(*
	DataWordInput1 AT %IB100 : ARRAY [0..15] OF WORD; 
	DataWordInput2 AT %IB132 : ARRAY [16..31] OF WORD; 
	DataWordInput3 AT %IB164 : ARRAY [32..47] OF WORD; 
	DataWordInput4 AT %IB196 : ARRAY [48..56] OF WORD; 
	DataWordOutput1 AT %QB100 : ARRAY [0..15] OF WORD; 
	DataWordOutput2 AT %QB132 : ARRAY [16..31] OF WORD; 
	DataWordOutput3 AT %QB164 : ARRAY [32..47] OF WORD; 
	DataWordOutput4 AT %QB196 : ARRAY [48..56] OF WORD; 
	*)
	Gateway_Q0_MODE_COMMAND_0 AT %QX100.0 : BOOL ;
	Gateway_Q0_MODE_COMMAND_1 AT %QX100.1 : BOOL ;
	Gateway_Q0_RESET AT %QX100.4 : BOOL;
	Gateway_Q0_RESTART AT %QX100.5 : BOOL;
	Gateway_Q0_STOP AT %QX100.7 : BOOL;
	Gateway_Q1_0 AT %QX101.0 : BOOL;
	Gateway_Q1_1 AT %QX101.1 : BOOL;
	Gateway_Q1_2 AT %QX101.2 : BOOL;
	Gateway_Q1_3 AT %QX101.3 : BOOL;
	Gateway_Q1_4 AT %QX101.4 : BOOL;
	Gateway_Gateway_Unit_2_Status AT %QB102 : BYTE;
	Gateway_Q3_0 AT %QX103.0 : BOOL;
	Gateway_Q3_1 AT %QX103.1 : BOOL;
	Gateway_Q3_2 AT %QX103.2 : BOOL;
	Gateway_Q3_3 AT %QX103.3 : BOOL;	
	

	ID1_StepData AT %QB114 : BYTE;
	ID1_Hold AT %QX115.0 : BOOL;
	ID1_SVON AT %QX115.1 : BOOL;
	ID1_Drive AT %QX115.2 : BOOL;
	ID1_Reset AT %QX115.3 : BOOL;
	ID1_Setup AT %QX115.4 : BOOL;
	

	ID2_StepData AT %QB134 : BYTE;
	ID2_Hold AT %QX135.0 : BOOL;
	ID2_SVON AT %QX135.1 : BOOL;
	ID2_Drive AT %QX135.2 : BOOL;
	ID2_Reset AT %QX135.3 : BOOL;
	ID2_Setup AT %QX135.4 : BOOL;


	ID3_StepData AT %QB154 : BYTE;
	ID3_Hold AT %QX155.0 : BOOL;
	ID3_SVON AT %QX155.1 : BOOL;
	ID3_Drive AT %QX155.2 : BOOL;
	ID3_Reset AT %QX155.3 : BOOL;
	ID3_Setup AT %QX155.4 : BOOL;
	
	
	ID4_StepData AT %QB174 : BYTE;
	ID4_Hold AT %QX175.0 : BOOL;
	ID4_SVON AT %QX175.1 : BOOL;
	ID4_Drive AT %QX175.2 : BOOL;
	ID4_Reset AT %QX175.3 : BOOL;
	ID4_Setup AT %QX175.4 : BOOL;
	

	ID5_StepData AT %QB194 : BYTE;
	ID5_Hold AT %QX195.0 : BOOL;
	ID5_SVON AT %QX195.1 : BOOL;
	ID5_Drive AT %QX195.2 : BOOL;
	ID5_Reset AT %QX195.3 : BOOL;
	ID5_Setup AT %QX195.4 : BOOL;
	
	byte0 : BYTE;
	byte1 : BYTE;
	byte2 : BYTE;
	byte3 : BYTE;
	
	bit14_0 : BOOL;
	bit14_1 : BOOL;
	bit14_2 : BOOL;
	bit14_3 : BOOL;
	bit14_4 : BOOL;
	bit14_5 : BOOL;
	
	bit15_0 : BOOL;
	bit15_1 : BOOL;
	bit15_2 : BOOL;
	bit15_3 : BOOL;
	bit15_4 : BOOL; 
	
	bit34_0 : BOOL;
	bit34_1 : BOOL;
	bit34_2 : BOOL;
	bit34_3 : BOOL;
	bit34_4 : BOOL;
	bit34_5 : BOOL;
	
	bit35_0 : BOOL;
	bit35_1 : BOOL;
	bit35_2 : BOOL;
	bit35_3 : BOOL;
	bit35_4 : BOOL; 
	
	bit54_0 : BOOL;
	bit54_1 : BOOL;
	bit54_2 : BOOL;
	bit54_3 : BOOL;
	bit54_4 : BOOL;
	bit54_5 : BOOL;
	
	bit55_0 : BOOL;
	bit55_1 : BOOL;
	bit55_2 : BOOL;
	bit55_3 : BOOL;
	bit55_4 : BOOL; 
	
	bit74_0 : BOOL;
	bit74_1 : BOOL;
	bit74_2 : BOOL;
	bit74_3 : BOOL;
	bit74_4 : BOOL;
	bit74_5 : BOOL;
	
	bit75_0 : BOOL;
	bit75_1 : BOOL;
	bit75_2 : BOOL;
	bit75_3 : BOOL;
	bit75_4 : BOOL; 
	
	bit94_0 : BOOL;
	bit94_1 : BOOL;
	bit94_2 : BOOL;
	bit94_3 : BOOL;
	bit94_4 : BOOL;
	bit94_5 : BOOL;
	
	bit95_0 : BOOL;
	bit95_1 : BOOL;
	bit95_2 : BOOL;
	bit95_3 : BOOL;
	bit95_4 : BOOL; 	
	
	ID1_I0_MODE_COMMAND_0 AT %IX100.0 : BOOL :=0;
	ID1_I0_MODE_COMMAND_1 AT %IX100.1 : BOOL:=0;
	ID1_I0_READY AT %IX100.4 : BOOL;
	ID1_I0_ALARM AT %IX100.5 : BOOL;
	ID1_I0_INITIAL AT %IX100.6 : BOOL;
	ID1_I0_COMMUNICATING AT %IX100.7 : BOOL;
	ID1_I1_0 AT %IX101.0 : BOOL;
	ID1_I1_1 AT %IX101.1 : BOOL;
	ID1_I1_2 AT %IX101.2 : BOOL;
	ID1_I1_3 AT %IX101.3 : BOOL;
	ID1_I1_4 AT %IX101.4 : BOOL;
	ID1_I2_0 AT %IX102.0 : BOOL;
	ID1_I2_1 AT %IX102.1 : BOOL;
	ID1_I2_2 AT %IX102.2 : BOOL;
	ID1_I2_3 AT %IX102.3 : BOOL;
	ID1_I2_4 AT %IX102.4 : BOOL;

	ID1_I3_0 AT %IX103.0 : BOOL;
	ID1_I3_1 AT %IX103.1 : BOOL;
	
	ID1_I32_0 AT %IX132.0 : BOOL;
	ID1_I32_1 AT %IX132.1 : BOOL;
	ID1_I33_0 AT %IX133.0 : BOOL;
	ID1_I33_1 AT %IX133.1 : BOOL;
(*-----------------------------------------------------------*)

	iTest15: SINT;
	iTest16: SINT;
	
	bTest1 : BOOL;
	bTest2 : BOOL;
	bTest3 : BOOL;
	bTest4 : BOOL;
	bTest5 : BOOL;
	bTest6 : BOOL;
	bTest7 : BOOL;
	bTest8 : BOOL;
	bTest9 : BOOL;
	bTest10 : BOOL;
	bTest11 : BOOL;
	bTest12 : BOOL;
	bTest13 : BOOL;
	bTest14 : BOOL;
	
	StepData1 : BYTE;
	StepData2 : BYTE;
	StepData3 : BYTE;
	StepData4 : BYTE;
	StepData5 : BYTE;
	
	star :BOOL;
	hom : BOOL;

	reset: BOOL;
	
	ID1_ALARM AT%IX115.7 : BOOL;
	ID2_ALARM AT%IX135.7 : BOOL;
	ID3_ALARM AT%IX155.7 : BOOL;
	ID4_ALARM AT%IX175.7 : BOOL;
	ID5_ALARM AT%IX195.7 : BOOL;
	
	ID1_SVRE AT%IX115.1 : BOOL;
	ID2_SVRE AT%IX135.1 : BOOL;
	ID3_SVRE AT%IX155.1 : BOOL;
	ID4_SVRE AT%IX175.1 : BOOL;
	ID5_SVRE AT%IX195.1 : BOOL;
	
	ID1_INP AT%IX115.3 : BOOL;
	ID2_INP AT%IX135.3 : BOOL;
	ID3_INP AT%IX155.3 : BOOL;
	ID4_INP AT%IX175.3 : BOOL;
	ID5_INP AT%IX195.3 : BOOL;
	
	PROSES: STRING;
	STAGE: INT;
	
	PROCESS: INT;
	START_PROCESS: BOOL;
	STEP_DATAS: INT;
	PROCESS_DELAY: TIME :=T#300MS;
	FUKUDA_RUNNING: BOOL :=FALSE;
	ACTIVE_STEPDATA : BYTE;
	//ACTIVE_ID: INT :=1;
	TMR1: TON;
	TMR2: TON;
	TMR3: TON;
	TMR4: TON;
	TMR5: TON;
	TMR6: TON;
	TMR10: Ton;
	TMR11: TON;
	TMR12: TON;
	TMR13: TON;
	TMR14: TON;
	TMR20: TON;
	TMR21: TON;
	TMR22: TON;
	TMR23: TON;
	TMR30: TON;
	TMR31: TON;
	TMR32: TON;
	TMR33: TON;
	TMR40: TON;
	TMR41: TON;
	TMR42: TON;
	TMR43: TON;
	TMR50: TON;
	TMR51: TON;
	TMR52: TON;
	TMR53: TON;
	
	
	TMR101: TON;
	TMR102: TON;
	TMR103: TON;
	TMR104: TON;
	TMR105: TON;
	TMR106: TON;
	ID5: INT;
	TMR7: Ton;
	TMR_RES_CARTSN: TOF;
	TMR_ACTIVATE_RESET: TON;
END_VAR


PROCESS_DELAY:= T#400MS;
IF 	INPUT_VAR.ACTIVE_ID >=0 THEN
STEP_DATA_1:=STEP_DATA_1+1;

IF STEP_DATA_2>=5 THEN
	STEP_DATA_2:=STEP_DATA_2+1;
END_IF

STEP_DATA_3:=STEP_DATA_3+1;	
END_IF


IF NOT INPUT_VAR.FUKUDA_HOME THEN //fukuda_running THEN
	IF  ID1_SVRE AND ID2_SVRE  AND  ID3_SVRE AND  ID4_SVRE AND  ID5_SVRE THEN
		TMR1(IN:=TRUE,PT:=T#0.5S);
		TMR4(IN:=TRUE,PT:=T#3S);
		TMR5(IN:=TRUE,PT:=T#3.5S);
		TMR6(IN:=TRUE,PT:=T#25S);
		IF ID1_SVRE THEN
			ID1_SETUP :=TMR5.Q;
		ELSE
			ID1_SVON :=TRUE;	
		END_IF

		IF ID2_SVRE THEN
			ID2_SETUP :=TMR1.Q;
		ELSE
			ID2_SVON :=TRUE;	
		END_IF
	
		IF ID3_SVRE THEN
		ID3_SETUP :=TMR4.Q;
		ELSE
			ID3_SVON :=TRUE;	
		END_IF
		CASE INPUT_VAR.I_CURRENT_TRANSACTION.TRANSPORT_INDEX OF
		1:
			TMR2(IN:=TRUE,PT:=T#1S);
			IF ID4_SVRE THEN
				ID4_SETUP :=TMR2.Q;
			ELSE
				ID4_SVON :=TRUE;	
			END_IF
		2:
			TMR3(IN:=TRUE,PT:=T#1.5S);
			IF ID5_SVRE THEN
				ID5_SETUP :=TMR3.Q;
			ELSE
				ID5_SVON :=TRUE;	
			END_IF
		END_CASE

	//IF TMR6.Q THEN
	IF ID1_INP AND ID2_INP AND ID3_INP AND (ID4_INP OR ID5_INP) THEN
		ID1_SETUP :=FALSE;
		ID2_SETUP :=FALSE;
		ID3_SETUP :=FALSE;
		ID4_SETUP :=FALSE;
		ID5_SETUP :=FALSE;
	
		TMR1(IN:=FALSE);
		TMR2(IN:=FALSE);
		TMR3(IN:=FALSE);
		TMR4(IN:=FALSE);
		TMR5(IN:=FALSE);
	//ACTIVE_ID:=1;
	//FUKUDA_RUNNING:=TRUE;
		INPUT_VAR.FUKUDA_HOME:=TRUE;
	END_IF
	
	ELSE
				
	ID1_SVON :=TRUE;
	ID2_SVON :=TRUE;
	ID3_SVON :=TRUE;
	ID4_SVON :=TRUE;
	ID5_SVON :=TRUE;

	END_IF
ELSE
	TMR6(IN:=FALSE);

	CASE INPUT_VAR.ACTIVE_ID OF
	0:
		INPUT_VAR.I_CASE:=INPUT_VAR.I_CASE+1;
		//INPUT_VAR.I_FUKUDA_RUNNING:=FALSE;
		INPUT_VAR.ACTIVE_ID:=6;
		
	1:
		IF STEP_DATA_1 = 0 THEN
			INPUT_VAR.ACTIVE_ID:=2;
		ELSE
			IF ID1_ALARM THEN
				Reset := TRUE;
				TMR10(IN:=TRUE,PT:= PROCESS_DELAY);
				IF TMR10.Q THEN
					Reset := FALSE;
				END_IF
			ELSE
				ID1_StepData :=STEP_DATA_1;
				ID1_Drive := FALSE;
				TMR11(IN:=TRUE,PT:= PROCESS_DELAY);
				IF TMR11.Q THEN
					IF ID1_INP THEN
					ID1_Drive := TRUE;
					TMR12(IN:=TMR11.Q,PT:= PROCESS_DELAY);
					IF TMR12.Q THEN
						ID1_Drive := FALSE;
						INPUT_VAR.ACTIVE_ID:=2;
						TMR10(IN:=FALSE);
						TMR11(IN:=FALSE);
						TMR12(IN:=FALSE);
						INPUT_VAR.FUKUDA_HOME:=TRUE;
					END_IF
					END_IF
				END_IF
			END_IF
		END_IF
	//	INPUT_VAR.I_CASE:=INPUT_VAR.I_CASE+1;
		//INPUT_VAR.I_FUKUDA_RUNNING:=FALSE;
	2:
		IF STEP_DATA_2 = 0 THEN
			INPUT_VAR.ACTIVE_ID:=3;
		ELSE
			
			IF ID2_ALARM THEN
				Reset := TRUE;
				TMR20(IN:=TRUE,PT:= PROCESS_DELAY);
				IF TMR20.Q THEN
					Reset := FALSE;
				END_IF
			ELSE
			ID2_StepData :=STEP_DATA_2;
			TMR21(IN:=TRUE,PT:= PROCESS_DELAY);
			IF TMR21.Q THEN
				ID2_Drive := TRUE;
				TMR22(IN:=TMR21.Q,PT:= PROCESS_DELAY);
				IF TMR22.Q THEN
				IF ID2_INP THEN
					ID2_Drive := FALSE;
					INPUT_VAR.ACTIVE_ID:=3;
					TMR20(IN:=FALSE);
					TMR21(IN:=FALSE);
					TMR22(IN:=FALSE);
				END_IF
				END_IF
			END_IF
			END_IF
		END_IF
	3:
		IF STEP_DATA_3 = 0 THEN
			INPUT_VAR.ACTIVE_ID:=4;
		ELSE
			
		IF ID3_ALARM THEN
			Reset := TRUE;
			TMR30(IN:=START_PROCESS,PT:= PROCESS_DELAY);
			IF TMR30.Q THEN
				Reset := FALSE;
			END_IF
		ELSE
		
		ID3_StepData :=STEP_DATA_3;
		TMR31(IN:=TRUE,PT:= PROCESS_DELAY);
		IF TMR31.Q THEN
			ID3_DRIVE := TRUE;	
			TMR32(IN:=TMR31.Q,PT:= PROCESS_DELAY);
			
			IF TMR32.Q THEN
				IF  ID3_INP THEN
				ID3_Drive := FALSE;
				INPUT_VAR.ACTIVE_ID:=4;
				TMR30(IN:=FALSE);
				TMR31(IN:=FALSE);
				TMR32(IN:=FALSE);
				END_IF
			END_IF
		END_IF
		END_IF
	END_IF
4:
		IF STEP_DATA_4 = 0 THEN
			INPUT_VAR.ACTIVE_ID:=5;
		ELSE
			IF ID4_ALARM THEN
				Reset := TRUE;
				TMR40(IN:=TRUE,PT:= PROCESS_DELAY);
				IF TMR40.Q THEN
					Reset := FALSE;
				END_IF
			ELSE
			
			ID4_StepData :=STEP_DATA_4;
			TMR41(IN:=TRUE,PT:= PROCESS_DELAY);
			IF TMR41.Q THEN
				ID4_Drive := TRUE;
				TMR42(IN:=TMR41.Q,PT:= PROCESS_DELAY);
				
				IF TMR42.Q THEN
					ID4_Drive := FALSE;
					INPUT_VAR.ACTIVE_ID:=5;
					TMR40(IN:=FALSE);
					TMR41(IN:=FALSE);
					TMR42(IN:=FALSE);
				END_IF
			END_IF
			END_IF
		END_IF
	5:
		IF STEP_DATA_5 = 0 THEN
			INPUT_VAR.ACTIVE_ID:=0;
		ELSE
			
			IF ID5_ALARM THEN
				Reset := TRUE;
				TMR50(IN:=TRUE,PT:= PROCESS_DELAY);
				IF TMR50.Q THEN
					Reset := FALSE;
				END_IF
			ELSE
			
			ID5_StepData :=STEP_DATA_5;
			TMR51(IN:=TRUE,PT:= PROCESS_DELAY);
			IF TMR51.Q THEN
				ID5_Drive := TRUE;	
				TMR52(IN:=TMR51.Q,PT:= PROCESS_DELAY);
				IF TMR52.Q THEN
					ID5_Drive := FALSE;
					INPUT_VAR.ACTIVE_ID:=0;
					TMR50(IN:=FALSE);
					TMR51(IN:=FALSE);
					TMR52(IN:=FALSE);
			
				END_IF
			END_IF
			END_IF
		END_IF
		
END_CASE 

	//START_PROCESS := FALSE;
END_IF
TMR7(IN:=reset,PT:= T#1S);
IF  tmr7.Q THEN
	reset:=FALSE;
END_IF
IF ID1_ALARM OR ID2_ALARM OR ID3_ALARM OR ID4_ALARM OR ID5_ALARM THEN
			reset:=TRUE;
			ELSE
				reset:=FALSE;
			END_IF
IF reset THEN
	ID1_Reset := TRUE;
	ID2_Reset := TRUE;
	ID3_Reset := TRUE;
	ID4_Reset := TRUE;
	ID5_Reset := TRUE;
	TMR_ACTIVATE_RESET(IN:=TRUE,PT:=T#10S);
	IF TMR_ACTIVATE_RESET.Q THEN
		TMR_RES_CARTSN(IN:=TRUE,PT:=T#0.5S);
	END_IF
	
ELSE
	TMR_ACTIVATE_RESET(IN:=FALSE);
	TMR_RES_CARTSN(IN:=FALSE);
	ID1_Reset := FALSE;
	ID2_Reset := FALSE;
	ID3_Reset := FALSE;
	ID4_Reset := FALSE;
	ID5_Reset := FALSE;
END_IF
INPUT_VAR.O_RESET_CARTESSIAN := TMR_RES_CARTSN.Q;

END_PROGRAM

// ---- POUs/FUKUDA/RETURN_FUKUDA.TcPOU
PROGRAM RETURN_FUKUDA
VAR_INPUT

END_VAR

VAR
	TMR_DELAY: TON;
END_VAR

CASE INPUT_VAR.I_CASE OF
0: //standby near lotbox
	IF INPUT_VAR.ACTIVE_ID=6 THEN
		INPUT_VAR.ACTIVE_ID:=1;
	END_IF

	CASE INPUT_VAR.I_CURRENT_TRANSACTION.TRANSPORT_INDEX OF
		2 : 
			INPUT_VAR.O_STOPPER_TRANSFER_B:=FALSE;			
			FUKUDA_MOVE(STEP_DATA_1:=3,
				STEP_DATA_2:=1,
				STEP_DATA_3:=12,
				STEP_DATA_4:=0,
				STEP_DATA_5:=1);
		1 : 
			INPUT_VAR.O_STOPPER_TRANSFER_A:=FALSE;
			FUKUDA_MOVE(STEP_DATA_1:=3,
				STEP_DATA_2:=1,
				STEP_DATA_3:=12,
				STEP_DATA_4:=1,
				STEP_DATA_5:=0);
	END_CASE			
	input_var.O_VACUUM_On:=FALSE;
	input_var.O_VACUUM_OFF:=FALSE;	
	TMR_DELAY(IN:=FALSE);

1://ready for picking up
	IF INPUT_VAR.ACTIVE_ID=6 THEN
		INPUT_VAR.ACTIVE_ID:=1;
	END_IF

		CASE INPUT_VAR.I_CURRENT_TRANSACTION.TRANSPORT_INDEX OF
		1:
			INPUT_VAR.I_RETURN_DONE_A:=FALSE;
		
		2:
			INPUT_VAR.I_RETURN_DONE_B:=FALSE;
	END_CASE
	FUKUDA_MOVE(STEP_DATA_1:=3,
				STEP_DATA_2:=1,
				STEP_DATA_3:=13,
				STEP_DATA_4:=0,
				STEP_DATA_5:=0);	
			
2://ready for picking up
	IF INPUT_VAR.ACTIVE_ID=6 THEN
		INPUT_VAR.ACTIVE_ID:=1;
	END_IF

	CASE INPUT_VAR.I_CURRENT_TRANSACTION.TRANSPORT_INDEX OF
	1:		
		IF INPUT_VAR.I_FUKUDA_TRANSFER_AT_BACK_A THEN
		FUKUDA_MOVE(STEP_DATA_1:=INPUT_VAR.I_CURRENT_TRANSACTION.TRANSPORT_INDEX+4,
				STEP_DATA_2:=1,
				STEP_DATA_3:=11,
				STEP_DATA_4:=0,
				STEP_DATA_5:=0);
		END_IF
	2:
		IF INPUT_VAR.I_FUKUDA_TRANSFER_AT_BACK_B THEN
		FUKUDA_MOVE(STEP_DATA_1:=INPUT_VAR.I_CURRENT_TRANSACTION.TRANSPORT_INDEX+4,
				STEP_DATA_2:=1,
				STEP_DATA_3:=11,
				STEP_DATA_4:=0,
				STEP_DATA_5:=0);
	END_IF
	END_CASE
	
		
3://placing onto fukuda transport
	IF INPUT_VAR.ACTIVE_ID=6 THEN
		INPUT_VAR.ACTIVE_ID:=1;
	END_IF

	FUKUDA_MOVE(STEP_DATA_1:=INPUT_VAR.I_CURRENT_TRANSACTION.TRANSPORT_INDEX+4,
				STEP_DATA_2:=2,
				STEP_DATA_3:=11,
				STEP_DATA_4:=0,
				STEP_DATA_5:=0);
	
4://ready for picking up
	IF INPUT_VAR.ACTIVE_ID=6 THEN
		INPUT_VAR.ACTIVE_ID:=1;
	END_IF
	
	FUKUDA_MOVE(STEP_DATA_1:=INPUT_VAR.I_CURRENT_TRANSACTION.TRANSPORT_INDEX+4,
				STEP_DATA_2:=6,
				STEP_DATA_3:=11,
				STEP_DATA_4:=0,
				STEP_DATA_5:=0);

5://gripping position
	IF INPUT_VAR.ACTIVE_ID=6 THEN
		INPUT_VAR.ACTIVE_ID:=1;
	END_IF
	
	IF NOT input_var.I_VACUUM_On THEN
		FUKUDA_MOVE(STEP_DATA_1:=INPUT_VAR.I_CURRENT_TRANSACTION.TRANSPORT_INDEX+4,
				STEP_DATA_2:=2,
				STEP_DATA_3:=12,
				STEP_DATA_4:=0,
				STEP_DATA_5:=0);
	ELSE
		input_var.O_VACUUM_On:=TRUE;
		input_var.O_VACUUM_OFF:=FALSE;
	END_IF
	
				
6://vacuum position 
	IF INPUT_VAR.ACTIVE_ID=6 THEN
		INPUT_VAR.ACTIVE_ID:=1;
	END_IF
	
	FUKUDA_MOVE(STEP_DATA_1:=INPUT_VAR.I_CURRENT_TRANSACTION.STATION_NUMBER_RETURN,
				STEP_DATA_2:=3,
				STEP_DATA_3:=INPUT_VAR.I_CURRENT_TRANSACTION.JIG_INDEX_RETURN,
				STEP_DATA_4:=0,
				STEP_DATA_5:=0);
				
7://vacuum position 
	IF INPUT_VAR.ACTIVE_ID=6 THEN
		INPUT_VAR.ACTIVE_ID:=1;
	END_IF
	TMR_DELAY(IN:=TRUE,PT:=T#1S);
	IF TMR_DELAY.Q THEN
			FUKUDA_MOVE(STEP_DATA_1:=INPUT_VAR.I_CURRENT_TRANSACTION.STATION_NUMBER_RETURN,
				STEP_DATA_2:=3,
				STEP_DATA_3:=14,
				STEP_DATA_4:=0,
				STEP_DATA_5:=0);
	END_IF
				
8://vacuum position 
	IF INPUT_VAR.ACTIVE_ID=6 THEN
		INPUT_VAR.ACTIVE_ID:=1;
	END_IF
	TMR_DELAY(IN:=FALSE);
	FUKUDA_MOVE(STEP_DATA_1:=INPUT_VAR.I_CURRENT_TRANSACTION.STATION_NUMBER_RETURN,
				STEP_DATA_2:=7,
				STEP_DATA_3:=16,
				STEP_DATA_4:=0,
				STEP_DATA_5:=0);
				
9://vacuum position 
	IF INPUT_VAR.ACTIVE_ID=6 THEN
		INPUT_VAR.ACTIVE_ID:=1;
	END_IF
	
	FUKUDA_MOVE(STEP_DATA_1:=INPUT_VAR.I_CURRENT_TRANSACTION.STATION_NUMBER_RETURN,
				STEP_DATA_2:=8,
				STEP_DATA_3:=INPUT_VAR.I_CURRENT_TRANSACTION.JIG_INDEX_RETURN,
				STEP_DATA_4:=0,
				STEP_DATA_5:=0);
10: //standby near lotbox
	
	IF INPUT_VAR.ACTIVE_ID=6 THEN
		INPUT_VAR.ACTIVE_ID:=1;
	END_IF

	IF input_var.I_VACUUM_ON THEN
		FUKUDA_MOVE(STEP_DATA_1:=INPUT_VAR.I_CURRENT_TRANSACTION.STATION_NUMBER_RETURN,
				STEP_DATA_2:=4,
				STEP_DATA_3:=INPUT_VAR.I_CURRENT_TRANSACTION.JIG_INDEX_RETURN,
				STEP_DATA_4:=0,
				STEP_DATA_5:=0);
	ELSE
		input_var.O_VACUUM_ON:=FALSE;
		input_var.O_VACUUM_OFF:=TRUE;			
	END_IF
	
				
11://vacuum position 
	IF INPUT_VAR.ACTIVE_ID=6 THEN
		INPUT_VAR.ACTIVE_ID:=1;
	END_IF
	FUKUDA_MOVE(STEP_DATA_1:=INPUT_VAR.I_CURRENT_TRANSACTION.STATION_NUMBER_RETURN,
				STEP_DATA_2:=1,
				STEP_DATA_3:=INPUT_VAR.I_CURRENT_TRANSACTION.JIG_INDEX_RETURN,
				STEP_DATA_4:=0,
				STEP_DATA_5:=0);
	IF INPUT_VAR.ACTIVE_ID=3 THEN
		input_var.O_VACUUM_ON:=FALSE;
		input_var.O_VACUUM_OFF:=FALSE;	
	END_IF
	
12://vacuum position 
	IF INPUT_VAR.ACTIVE_ID=6 THEN
		INPUT_VAR.ACTIVE_ID:=1;
	END_IF
	FUKUDA_MOVE(STEP_DATA_1:=0,
				STEP_DATA_2:=1,
				STEP_DATA_3:=4,
				STEP_DATA_4:=0,
				STEP_DATA_5:=0);				
		
100:
	
	input_var.O_VACUUM_On:=FALSE;
	input_var.O_VACUUM_OFF:=FALSE;
END_CASE 
IF INPUT_VAR.I_CASE=13 THEN
			CASE INPUT_VAR.I_CURRENT_TRANSACTION.TRANSPORT_INDEX OF
		1:
			INPUT_VAR.I_RETURN_DONE_A:=TRUE;
		
		2:
			INPUT_VAR.I_RETURN_DONE_B:=TRUE;
	END_CASE
	IF INPUT_VAR.I_RETURN_DONE_A OR INPUT_VAR.I_RETURN_DONE_B THEN
		FLAG_VAR.ALLOW_EXECUTE_RETURN_FUKUDA:=FALSE;
		INPUT_VAR.I_CASE:=100;
	END_IF
END_IF

END_PROGRAM

// ---- POUs/ROBOT/LOADER_RS4.TcPOU
PROGRAM LOADER_RS4
VAR

	TMR10: TON;
	TMR8: TON;
	TMR9: TON;
	TMR7: TON;
	TMR3: TON;
	POSITION_CHANGED: BOOL;
	START_MOVE: TP;
	TMR1: TON;
	TP2: TP;
	START_ROBOT: TP;
	TMR2: TON;
	GO_ROBOT: BOOL;
	TP_COUNT: R_TRIG;
	CNT_INC: CTU;
	VAL: INT;
	ROT_START:R_TRIG;
	RESET_POSITION: BOOL;
	RES_POS: TON;
	CNT_CYCLE: CTU;
	START_ROTATE: R_TRIG;
END_VAR


IF LOADER_RS4_VAR.I_LOADER_RS4_ENABLE THEN
IF LOADER_RS4_VAR.IX_LOADER_RS4_GRIPPER_1 THEN
	LOADER_RS4_VAR.O_LOADER_RS4_GRIPPER_CLOSE_1:=TRUE;
	LOADER_RS4_VAR.O_LOADER_RS4_GRIPPER_OPEN_1:=FALSE;
ELSE
	LOADER_RS4_VAR.O_LOADER_RS4_GRIPPER_CLOSE_1:=FALSE;
	LOADER_RS4_VAR.O_LOADER_RS4_GRIPPER_OPEN_1:=TRUE;
END_IF

IF LOADER_RS4_VAR.IX_LOADER_RS4_GRIPPER_2 THEN
	LOADER_RS4_VAR.O_LOADER_RS4_GRIPPER_CLOSE_2:=TRUE;
	LOADER_RS4_VAR.O_LOADER_RS4_GRIPPER_OPEN_2:=FALSE;
ELSE
	LOADER_RS4_VAR.O_LOADER_RS4_GRIPPER_CLOSE_2:=FALSE;
	LOADER_RS4_VAR.O_LOADER_RS4_GRIPPER_OPEN_2:=TRUE;
END_IF

IF LOADER_RS4_VAR.IX_LOADER_RS4_GRIPPER_3 THEN
	LOADER_RS4_VAR.O_LOADER_RS4_GRIPPER_CLOSE_3:=TRUE;
	LOADER_RS4_VAR.O_LOADER_RS4_GRIPPER_OPEN_3:=FALSE;
ELSE
	LOADER_RS4_VAR.O_LOADER_RS4_GRIPPER_CLOSE_3:=FALSE;
	LOADER_RS4_VAR.O_LOADER_RS4_GRIPPER_OPEN_3:=TRUE;
END_IF

IF LOADER_RS4_VAR.IX_LOADER_RS4_GRIPPER_4 THEN
	LOADER_RS4_VAR.O_LOADER_RS4_GRIPPER_CLOSE_4:=TRUE;
	LOADER_RS4_VAR.O_LOADER_RS4_GRIPPER_OPEN_4:=FALSE;
ELSE
	LOADER_RS4_VAR.O_LOADER_RS4_GRIPPER_CLOSE_4:=FALSE;
	LOADER_RS4_VAR.O_LOADER_RS4_GRIPPER_OPEN_4:=TRUE;
END_IF

IF LOADER_RS4_VAR.IX_LOADER_RS4_GRIPPER_EXT_1 THEN
	LOADER_RS4_VAR.O_LOADER_RS4_GRIPPER_EXT_DOWN_1:=TRUE;
	LOADER_RS4_VAR.O_LOADER_RS4_GRIPPER_EXT_UP_1:=FALSE;
ELSE
	LOADER_RS4_VAR.O_LOADER_RS4_GRIPPER_EXT_DOWN_1:=FALSE;
	LOADER_RS4_VAR.O_LOADER_RS4_GRIPPER_EXT_UP_1:=TRUE;
END_IF


IF LOADER_RS4_VAR.IX_LOADER_RS4_GRIPPER_EXT_2 THEN
	LOADER_RS4_VAR.O_LOADER_RS4_GRIPPER_EXT_DOWN_2:=TRUE;
	LOADER_RS4_VAR.O_LOADER_RS4_GRIPPER_EXT_UP_2:=FALSE;
ELSE
	LOADER_RS4_VAR.O_LOADER_RS4_GRIPPER_EXT_DOWN_2:=FALSE;
	LOADER_RS4_VAR.O_LOADER_RS4_GRIPPER_EXT_UP_2:=TRUE;
END_IF


IF LOADER_RS4_VAR.IX_LOADER_RS4_GRIPPER_EXT_3 THEN
	LOADER_RS4_VAR.O_LOADER_RS4_GRIPPER_EXT_DOWN_3:=TRUE;
	LOADER_RS4_VAR.O_LOADER_RS4_GRIPPER_EXT_UP_3:=FALSE;
ELSE
	LOADER_RS4_VAR.O_LOADER_RS4_GRIPPER_EXT_DOWN_3:=FALSE;
	LOADER_RS4_VAR.O_LOADER_RS4_GRIPPER_EXT_UP_3:=TRUE;
END_IF


IF LOADER_RS4_VAR.IX_LOADER_RS4_GRIPPER_EXT_4 THEN
	LOADER_RS4_VAR.O_LOADER_RS4_GRIPPER_EXT_DOWN_4:=TRUE;
	LOADER_RS4_VAR.O_LOADER_RS4_GRIPPER_EXT_UP_4:=FALSE;
ELSE
	LOADER_RS4_VAR.O_LOADER_RS4_GRIPPER_EXT_DOWN_4:=FALSE;
	LOADER_RS4_VAR.O_LOADER_RS4_GRIPPER_EXT_UP_4:=TRUE;
END_IF


CARRIER_INDEX:=INDEXING_2_VAR.CARRIER_INDEX;
LOADER_RS4_VAR.O_LOADER_RS4_SETMOTORON:=TRUE;
TMR1(IN:=LOADER_RS4_VAR.O_LOADER_RS4_SETMOTORON ,PT:=T#0.5S);
IF TMR1.Q THEN
	TP2(IN:=TMR1.Q,PT:=T#1S);
	LOADER_RS4_VAR.O_LOADER_RS4_STOP:=TP2.Q;
END_IF
IF LOADER_RS4_VAR.O_LOADER_RS4_SETMOTORON AND INDEXING_1_VAR.I_INDEXING_1_ROTATION_DONE AND INDEXING_1_VAR.I_INDEXING_1_HOME THEN
	IF LOADER_RS4_VAR.I_LOADER_RS4_READY OR LOADER_RS4_VAR.I_LOADER_RS4_RUNNING THEN
//EROOR OVERRIDE
		IF LOADER_RS4_VAR.I_LOADER_RS4_ERROR THEN
			TMR10(IN:=LOADER_RS4_VAR.I_LOADER_RS4_ERROR,PT:=T#1S);
			IF TMR10.Q THEN
				LOADER_RS4_VAR.O_LOADER_RS4_RESET :=TRUE;	
			ELSE
				LOADER_RS4_VAR.O_LOADER_RS4_RESET :=FALSE;
			END_IF
		END_IF 

		TMR8(IN:=INPUT_G6_VAR.O_G6_SELECT_FUKUDA_A,PT:=T#5S);
		TMR9(IN:=INPUT_G6_VAR.O_G6_START,PT:=T#2S);
		
//START FOR 1ST TIME			
		IF LOADER_RS4_VAR.I_LOADER_RS4_READY AND NOT LOADER_RS4_VAR.I_LOADER_RS4_ERROR AND NOT LOADER_RS4_VAR.I_LOADER_RS4_RUNNING THEN
			TMR7(IN:=INDEXING_1_VAR.I_INDEXING_1_ROTATION_DONE,PT:=T#1S);
			START_ROBOT(IN:=TMR7.Q,PT:=T#3S);
			LOADER_RS4_VAR.O_LOADER_RS4_START :=TMR7.Q;
			RESET_POSITION:=TRUE;
		ELSE
			TMR7(IN:=FALSE);
		END_IF
			IF LOADER_RS4_VAR.I_LOADER_RS4_RUNNING AND LOADER_RS4_VAR.I_LOADER_RS4_READY_TAKEUP THEN
			LOADER_RS4_VAR.O_LOADER_RS4_START :=FALSE ;
		END_IF
		
//STOP
		IF LOADER_RS4_VAR.I_LOADER_RS4_END_FUKUDA AND NOT LOADER_RS4_VAR.I_LOADER_RS4_READY AND NOT LOADER_RS4_VAR.I_LOADER_RS4_RUNNING THEN
			TMR8(IN:=FALSE);
			TMR9(IN:=FALSE);
			LOADER_RS4_VAR.O_LOADER_RS4_STOP :=TRUE;
		END_IF
			TMR2(IN:=LOADER_RS4_VAR.O_LOADER_RS4_STOP,PT:=T#1S);
		IF TMR2.Q THEN
			LOADER_RS4_VAR.I_LOADER_RS4_HANG:=FALSE;
			LOADER_RS4_VAR.O_LOADER_RS4_STOP:=FALSE;
			TMR1(IN:=FALSE);
		END_IF	
			
